C03611=1038.223,237.560,-108.650,170.961,41.926,157.985
C03612=1038.230,237.808,-108.678,170.964,41.928,157.986
C03613=1038.236,238.056,-108.706,170.967,41.929,157.986
C03614=1038.243,238.304,-108.734,170.970,41.930,157.987
C03615=1038.249,238.553,-108.763,170.972,41.931,157.987
C03616=1038.257,238.801,-108.791,170.975,41.933,157.988
C03617=1038.263,239.050,-108.819,170.978,41.934,157.988
C03618=1038.270,239.298,-108.848,170.981,41.935,157.988
C03619=1038.276,239.546,-108.876,170.983,41.936,157.989
C03620=1038.283,239.794,-108.904,170.987,41.937,157.989
C03621=1038.289,240.043,-108.933,170.989,41.938,157.990
C03622=1038.297,240.291,-108.961,170.992,41.940,157.990
C03623=1038.304,240.539,-108.990,170.994,41.941,157.990
C03624=1038.310,240.788,-109.018,170.998,41.942,157.991
C03625=1038.317,241.036,-109.047,171.000,41.943,157.991
C03626=1038.323,241.284,-109.076,171.003,41.945,157.992
C03627=1038.330,241.532,-109.103,171.005,41.946,157.992
C03628=1038.337,241.781,-109.133,171.009,41.947,157.993
C03629=1038.343,242.029,-109.162,171.012,41.949,157.993
C03630=1038.350,242.278,-109.190,171.014,41.950,157.994
C03631=1038.356,242.526,-109.219,171.016,41.951,157.994
C03632=1038.363,242.774,-109.247,171.020,41.952,157.994
C03633=1038.369,243.022,-109.276,171.022,41.954,157.995
C03634=1038.376,243.271,-109.304,171.025,41.955,157.995
C03635=1038.383,243.519,-109.333,171.028,41.956,157.996
C03636=1038.389,243.767,-109.362,171.031,41.958,157.996
C03637=1038.396,244.015,-109.391,171.033,41.959,157.997
C03638=1038.402,244.263,-109.420,171.037,41.960,157.997
C03639=1038.409,244.512,-109.448,171.040,41.962,157.998
C03640=1038.416,244.760,-109.477,171.042,41.963,157.998
C03641=1038.423,245.008,-109.505,171.045,41.964,157.999
C03642=1038.429,245.256,-109.534,171.048,41.965,157.999
C03643=1038.436,245.505,-109.564,171.051,41.966,157.999
C03644=1038.442,245.753,-109.593,171.053,41.968,158.000
C03645=1038.448,246.001,-109.622,171.057,41.969,158.001
C03646=1038.454,246.250,-109.651,171.059,41.970,158.001
C03647=1038.461,246.497,-109.679,171.062,41.972,158.001
C03648=1038.468,246.746,-109.709,171.065,41.973,158.002
C03649=1038.474,246.994,-109.738,171.068,41.974,158.002
C03650=1038.481,247.242,-109.767,171.070,41.976,158.003
C03651=1038.487,247.491,-109.796,171.074,41.977,158.003
C03652=1038.494,247.739,-109.825,171.077,41.979,158.004
C03653=1038.501,247.987,-109.854,171.079,41.980,158.004
C03654=1038.507,248.235,-109.883,171.083,41.981,158.005
C03655=1038.515,248.549,-109.920,171.085,41.983,158.005
C03656=1038.524,248.863,-109.957,171.089,41.985,158.006
C03657=1038.532,249.178,-109.993,171.092,41.986,158.006
C03658=1038.541,249.493,-110.030,171.096,41.988,158.007
C03659=1038.547,249.741,-110.059,171.100,41.989,158.007
C03660=1038.553,249.989,-110.088,171.102,41.991,158.008
C03661=1038.560,250.237,-110.119,171.105,41.992,158.008
C03662=1038.566,250.485,-110.148,171.108,41.994,158.009
C03663=1038.573,250.733,-110.177,171.111,41.995,158.009
C03664=1038.579,250.981,-110.206,171.114,41.996,158.010
C03665=1038.587,251.230,-110.235,171.117,41.998,158.010
C03666=1038.593,251.478,-110.264,171.119,41.998,158.011
C03667=1038.600,251.726,-110.294,171.123,42.000,158.011
C03668=1038.606,251.974,-110.323,171.126,42.001,158.012
C03669=1038.612,252.223,-110.352,171.129,42.003,158.012
C03670=1038.619,252.471,-110.381,171.132,42.004,158.013
C03671=1038.626,252.719,-110.411,171.134,42.005,158.013
C03672=1038.633,252.967,-110.439,171.138,42.007,158.014
C03673=1038.640,253.216,-110.469,171.140,42.008,158.014
C03674=1038.646,253.463,-110.499,171.144,42.009,158.015
C03675=1038.653,253.712,-110.528,171.146,42.011,158.015
C03676=1038.659,253.960,-110.557,171.149,42.012,158.016
C03677=1038.666,254.208,-110.586,171.152,42.013,158.016
C03678=1038.673,254.456,-110.616,171.155,42.015,158.016
C03679=1038.679,254.705,-110.645,171.159,42.016,158.017
C03680=1038.686,254.953,-110.675,171.161,42.018,158.017
C03681=1038.693,255.201,-110.704,171.165,42.018,158.018
C03682=1038.700,255.449,-110.733,171.167,42.020,158.018
C03683=1038.707,255.697,-110.763,171.171,42.021,158.019
C03684=1038.713,255.946,-110.792,171.173,42.023,158.019
C03685=1038.720,256.194,-110.821,171.176,42.024,158.020
C03686=1038.727,256.442,-110.852,171.179,42.025,158.020
C03687=1038.733,256.690,-110.881,171.182,42.027,158.021
C03688=1038.740,256.938,-110.911,171.186,42.028,158.021
C03689=1038.746,257.187,-110.940,171.188,42.029,158.022
C03690=1038.754,257.435,-110.970,171.192,42.031,158.022
C03691=1038.761,257.683,-110.998,171.194,42.032,158.023
C03692=1038.768,257.931,-111.028,171.198,42.033,158.023
C03693=1038.774,258.179,-111.057,171.200,42.034,158.024
C03694=1038.781,258.427,-111.088,171.204,42.036,158.024
C03695=1038.787,258.675,-111.117,171.206,42.037,158.025
C03696=1038.795,258.924,-111.147,171.210,42.038,158.025
C03697=1038.801,259.172,-111.176,171.212,42.040,158.026
C03698=1038.808,259.420,-111.206,171.216,42.041,158.026
C03699=1038.815,259.669,-111.235,171.219,42.043,158.027
C03700=1038.821,259.916,-111.265,171.222,42.044,158.027
C03701=1038.829,260.164,-111.295,171.225,42.045,158.027
C03702=1038.835,260.413,-111.324,171.228,42.046,158.028
C03703=1038.843,260.660,-111.354,171.232,42.048,158.029
C03704=1038.849,260.909,-111.383,171.234,42.049,158.029
C03705=1038.856,261.157,-111.413,171.238,42.050,158.029
C03706=1038.863,261.405,-111.443,171.240,42.052,158.030
C03707=1038.869,261.653,-111.472,171.244,42.053,158.030
C03708=1038.877,261.901,-111.502,171.246,42.055,158.031
C03709=1038.884,262.150,-111.532,171.250,42.056,158.032
C03710=1038.890,262.397,-111.563,171.253,42.058,158.032
C03711=1038.898,262.711,-111.600,171.256,42.059,158.033
C03712=1038.906,263.023,-111.638,171.261,42.061,158.033
C03713=1038.915,263.336,-111.676,171.265,42.063,158.034
C03714=1038.923,263.649,-111.713,171.268,42.064,158.034
C03715=1038.930,263.897,-111.744,171.272,42.066,158.035
C03716=1038.936,264.145,-111.774,171.275,42.067,158.036
C03717=1038.943,264.393,-111.804,171.278,42.069,158.036
C03718=1038.950,264.641,-111.834,171.281,42.070,158.037
C03719=1038.956,264.889,-111.865,171.284,42.072,158.037
C03720=1038.963,265.137,-111.895,171.287,42.073,158.038
C03721=1038.971,265.385,-111.925,171.291,42.075,158.038
C03722=1038.976,265.633,-111.955,171.293,42.076,158.039
C03723=1038.984,265.881,-111.985,171.297,42.077,158.039
C03724=1038.991,266.130,-112.015,171.300,42.079,158.040
C03725=1038.997,266.378,-112.046,171.303,42.080,158.040
C03726=1039.004,266.626,-112.076,171.307,42.082,158.041
C03727=1039.011,266.874,-112.106,171.309,42.083,158.041
C03728=1039.017,267.122,-112.136,171.313,42.085,158.042
C03729=1039.024,267.370,-112.166,171.316,42.086,158.042
C03730=1039.031,267.618,-112.197,171.319,42.088,158.043
C03731=1039.037,267.866,-112.227,171.323,42.089,158.043
C03732=1039.044,268.114,-112.257,171.325,42.091,158.044
C03733=1039.050,268.363,-112.288,171.329,42.092,158.044
C03734=1039.057,268.610,-112.317,171.332,42.093,158.045
C03735=1039.064,268.858,-112.349,171.335,42.095,158.045
C03736=1039.071,269.106,-112.379,171.339,42.096,158.046
C03737=1039.077,269.354,-112.409,171.341,42.098,158.046
C03738=1039.084,269.602,-112.440,171.345,42.099,158.047
C03739=1039.090,269.851,-112.470,171.348,42.101,158.048
C03740=1039.098,270.099,-112.501,171.351,42.102,158.048
C03741=1039.103,270.346,-112.531,171.355,42.104,158.049
C03742=1039.111,270.595,-112.562,171.357,42.106,158.049
C03743=1039.118,270.843,-112.592,171.361,42.107,158.050
C03744=1039.124,271.091,-112.623,171.365,42.109,158.050
C03745=1039.131,271.339,-112.654,171.367,42.110,158.051
C03746=1039.137,271.587,-112.684,171.371,42.111,158.051
C03747=1039.144,271.835,-112.715,171.374,42.113,158.052
C03748=1039.151,272.083,-112.745,171.377,42.114,158.052
C03749=1039.158,272.331,-112.776,171.381,42.116,158.053
C03750=1039.164,272.579,-112.807,171.384,42.118,158.054
C03751=1039.171,272.827,-112.837,171.387,42.119,158.054
C03752=1039.178,273.075,-112.868,171.391,42.121,158.055
C03753=1039.184,273.323,-112.899,171.394,42.122,158.055
C03754=1039.191,273.571,-112.929,171.397,42.124,158.056
C03755=1039.197,273.819,-112.960,171.401,42.125,158.056
C03756=1039.204,274.067,-112.991,171.404,42.127,158.057
C03757=1039.211,274.315,-113.022,171.407,42.129,158.057
C03758=1039.218,274.563,-113.053,171.411,42.130,158.058
C03759=1039.224,274.811,-113.084,171.414,42.131,158.059
C03760=1039.231,275.059,-113.114,171.417,42.133,158.059
C03761=1039.238,275.307,-113.145,171.421,42.135,158.060
C03762=1039.244,275.555,-113.176,171.424,42.136,158.060
C03763=1039.252,275.803,-113.207,171.427,42.138,158.061
C03764=1039.258,276.051,-113.238,171.430,42.139,158.061
C03765=1039.265,276.299,-113.269,171.434,42.141,158.062
C03766=1039.272,276.547,-113.300,171.437,42.143,158.063
C03767=1039.280,276.864,-113.340,171.442,42.145,158.063
C03768=1039.289,277.181,-113.380,171.445,42.147,158.064
C03769=1039.297,277.499,-113.418,171.450,42.148,158.065
C03770=1039.306,277.816,-113.458,171.454,42.150,158.065
C03771=1039.313,278.064,-113.490,171.458,42.152,158.066
C03772=1039.320,278.312,-113.521,171.461,42.154,158.067
C03773=1039.326,278.560,-113.552,171.465,42.155,158.067
C03774=1039.333,278.809,-113.583,171.468,42.157,158.068
C03775=1039.340,279.056,-113.614,171.471,42.159,158.068
C03776=1039.347,279.304,-113.645,171.475,42.160,158.069
C03777=1039.354,279.552,-113.677,171.478,42.162,158.069
C03778=1039.360,279.799,-113.708,171.481,42.164,158.070
C03779=1039.366,280.048,-113.739,171.485,42.165,158.071
C03780=1039.373,280.296,-113.770,171.489,42.167,158.071
C03781=1039.380,280.543,-113.801,171.491,42.168,158.072
C03782=1039.386,280.791,-113.833,171.495,42.170,158.072
C03783=1039.393,281.039,-113.864,171.499,42.172,158.073
C03784=1039.400,281.287,-113.896,171.502,42.173,158.074
C03785=1039.407,281.535,-113.927,171.505,42.175,158.074
C03786=1039.413,281.783,-113.959,171.509,42.177,158.075
C03787=1039.420,282.031,-113.990,171.513,42.179,158.075
C03788=1039.427,282.279,-114.022,171.516,42.180,158.076
C03789=1039.433,282.527,-114.053,171.520,42.181,158.076
C03790=1039.440,282.775,-114.084,171.523,42.184,158.077
C03791=1039.447,283.022,-114.116,171.526,42.185,158.078
C03792=1039.454,283.270,-114.147,171.530,42.187,158.078
C03793=1039.460,283.518,-114.179,171.534,42.188,158.079
C03794=1039.467,283.766,-114.210,171.536,42.190,158.080
C03795=1039.474,284.014,-114.242,171.540,42.192,158.080
C03796=1039.481,284.262,-114.273,171.544,42.194,158.081
C03797=1039.487,284.510,-114.304,171.548,42.195,158.081
C03798=1039.494,284.758,-114.336,171.551,42.197,158.082
C03799=1039.501,285.006,-114.368,171.555,42.199,158.083
C03800=1039.508,285.254,-114.400,171.558,42.200,158.083
C03801=1039.515,285.502,-114.431,171.561,42.202,158.084
C03802=1039.522,285.750,-114.463,171.565,42.203,158.084
C03803=1039.528,285.997,-114.494,171.569,42.205,158.085
C03804=1039.535,286.245,-114.526,171.572,42.207,158.086
C03805=1039.542,286.493,-114.558,171.576,42.209,158.086
C03806=1039.549,286.740,-114.589,171.580,42.210,158.087
C03807=1039.556,286.989,-114.621,171.583,42.212,158.087
C03808=1039.562,287.237,-114.653,171.586,42.214,158.088
C03809=1039.569,287.485,-114.685,171.590,42.216,158.089
C03810=1039.576,287.733,-114.716,171.594,42.217,158.089
C03811=1039.583,287.980,-114.748,171.597,42.219,158.090
C03812=1039.589,288.228,-114.781,171.601,42.221,158.091
C03813=1039.596,288.476,-114.812,171.604,42.222,158.091
C03814=1039.603,288.724,-114.844,171.608,42.224,158.092
C03815=1039.610,288.972,-114.876,171.611,42.226,158.092
C03816=1039.617,289.220,-114.907,171.615,42.228,158.093
C03817=1039.623,289.467,-114.940,171.619,42.230,158.094
C03818=1039.630,289.715,-114.972,171.623,42.231,158.094
C03819=1039.637,289.962,-115.004,171.626,42.233,158.095
C03820=1039.644,290.210,-115.035,171.630,42.235,158.096
C03821=1039.651,290.459,-115.068,171.633,42.237,158.096
C03822=1039.657,290.707,-115.100,171.637,42.239,158.097
C03823=1039.666,291.035,-115.143,171.642,42.241,158.098
C03824=1039.676,291.365,-115.185,171.647,42.243,158.099
C03825=1039.684,291.694,-115.228,171.652,42.246,158.099
C03826=1039.693,292.023,-115.271,171.657,42.248,158.100
C03827=1039.700,292.271,-115.303,171.660,42.250,158.101
C03828=1039.707,292.519,-115.335,171.664,42.252,158.102
C03829=1039.713,292.767,-115.367,171.668,42.254,158.102
C03830=1039.720,293.015,-115.399,171.671,42.255,158.103
C03831=1039.728,293.262,-115.431,171.675,42.257,158.104
C03832=1039.734,293.510,-115.464,171.678,42.259,158.104
C03833=1039.741,293.757,-115.496,171.682,42.261,158.105
C03834=1039.748,294.006,-115.528,171.686,42.263,158.106
C03835=1039.755,294.254,-115.561,171.689,42.264,158.106
C03836=1039.762,294.501,-115.593,171.693,42.266,158.107
C03837=1039.768,294.748,-115.626,171.697,42.268,158.107
C03838=1039.775,294.997,-115.657,171.701,42.270,158.108
C03839=1039.782,295.245,-115.690,171.705,42.272,158.109
C03840=1039.789,295.492,-115.722,171.708,42.274,158.109
C03841=1039.796,295.740,-115.755,171.712,42.275,158.110
C03842=1039.802,295.988,-115.788,171.716,42.277,158.111
C03843=1039.808,296.235,-115.821,171.720,42.279,158.112
C03844=1039.815,296.483,-115.853,171.723,42.281,158.112
C03845=1039.822,296.731,-115.886,171.727,42.283,158.113
C03846=1039.828,296.979,-115.919,171.731,42.285,158.114
C03847=1039.835,297.226,-115.952,171.735,42.287,158.114
C03848=1039.842,297.474,-115.984,171.739,42.289,158.115
C03849=1039.849,297.722,-116.017,171.743,42.291,158.116
C03850=1039.855,297.969,-116.050,171.746,42.293,158.116
C03851=1039.862,298.218,-116.083,171.750,42.295,158.117
C03852=1039.868,298.465,-116.115,171.754,42.297,158.118
C03853=1039.875,298.713,-116.148,171.758,42.299,158.118
C03854=1039.882,298.961,-116.181,171.762,42.301,158.119
C03855=1039.889,299.208,-116.214,171.765,42.303,158.120
C03856=1039.896,299.456,-116.247,171.769,42.305,158.121
C03857=1039.903,299.703,-116.279,171.773,42.307,158.121
C03858=1039.909,299.951,-116.312,171.777,42.309,158.122
C03859=1039.916,300.199,-116.345,171.781,42.311,158.123
C03860=1039.922,300.447,-116.378,171.785,42.313,158.123
C03861=1039.929,300.695,-116.412,171.789,42.315,158.124
C03862=1039.936,300.942,-116.444,171.792,42.317,158.125
C03863=1039.943,301.189,-116.477,171.796,42.319,158.126
C03864=1039.949,301.438,-116.510,171.800,42.321,158.126
C03865=1039.956,301.685,-116.543,171.804,42.323,158.127
C03866=1039.963,301.933,-116.576,171.808,42.325,158.128
C03867=1039.970,302.180,-116.609,171.811,42.327,158.128
C03868=1039.977,302.428,-116.642,171.815,42.329,158.129
C03869=1039.984,302.675,-116.675,171.819,42.331,158.130
C03870=1039.990,302.924,-116.708,171.823,42.333,158.131
C03871=1039.997,303.171,-116.742,171.827,42.335,158.131
C03872=1040.005,303.419,-116.774,171.831,42.337,158.132
C03873=1040.011,303.666,-116.807,171.835,42.339,158.133
C03874=1040.018,303.914,-116.841,171.838,42.341,158.133
C03875=1040.025,304.162,-116.874,171.843,42.343,158.134
C03876=1040.032,304.409,-116.907,171.847,42.345,158.135
C03877=1040.039,304.657,-116.940,171.851,42.348,158.136
C03878=1040.046,304.904,-116.973,171.855,42.350,158.136
C03879=1040.055,305.250,-117.020,171.860,42.353,158.137
C03880=1040.065,305.596,-117.066,171.866,42.355,158.138
C03881=1040.075,305.942,-117.112,171.871,42.358,158.139
C03882=1040.084,306.288,-117.159,171.877,42.361,158.140
C03883=1040.091,306.536,-117.193,171.882,42.363,158.141
C03884=1040.099,306.783,-117.225,171.885,42.365,158.142
C03885=1040.106,307.031,-117.259,171.889,42.367,158.143
C03886=1040.113,307.279,-117.292,171.893,42.369,158.143
C03887=1040.119,307.526,-117.325,171.897,42.371,158.144
C03888=1040.126,307.774,-117.359,171.901,42.373,158.145
C03889=1040.133,308.021,-117.393,171.905,42.375,158.146
C03890=1040.140,308.270,-117.426,171.910,42.377,158.146
C03891=1040.148,308.516,-117.459,171.914,42.380,158.147
C03892=1040.155,308.764,-117.493,171.917,42.382,158.148
C03893=1040.162,309.012,-117.526,171.921,42.384,158.149
C03894=1040.168,309.259,-117.559,171.925,42.386,158.149
C03895=1040.176,309.507,-117.593,171.930,42.388,158.150
C03896=1040.183,309.755,-117.627,171.934,42.390,158.151
C03897=1040.191,310.002,-117.660,171.938,42.392,158.152
C03898=1040.197,310.250,-117.693,171.942,42.394,158.152
C03899=1040.204,310.497,-117.727,171.947,42.396,158.153
C03900=1040.211,310.745,-117.760,171.951,42.398,158.154
C03901=1040.219,310.993,-117.794,171.955,42.401,158.155
C03902=1040.226,311.240,-117.828,171.958,42.403,158.155
C03903=1040.233,311.488,-117.862,171.962,42.405,158.156
C03904=1040.240,311.735,-117.895,171.967,42.407,158.157
C03905=1040.248,311.982,-117.929,171.971,42.409,158.158
C03906=1040.254,312.231,-117.962,171.975,42.411,158.159
C03907=1040.261,312.478,-117.997,171.979,42.413,158.159
C03908=1040.268,312.726,-118.031,171.984,42.416,158.160
C03909=1040.274,312.973,-118.065,171.988,42.418,158.161
C03910=1040.281,313.221,-118.098,171.992,42.420,158.162
C03911=1040.288,313.469,-118.133,171.996,42.423,158.163
C03912=1040.295,313.716,-118.167,172.000,42.425,158.163
C03913=1040.301,313.963,-118.201,172.005,42.427,158.164
C03914=1040.309,314.211,-118.235,172.009,42.430,158.165
C03915=1040.315,314.459,-118.270,172.013,42.432,158.166
C03916=1040.322,314.706,-118.304,172.017,42.434,158.167
C03917=1040.330,314.953,-118.338,172.022,42.436,158.167
C03918=1040.336,315.201,-118.372,172.026,42.439,158.168
C03919=1040.343,315.448,-118.406,172.030,42.441,158.169
C03920=1040.349,315.696,-118.440,172.034,42.443,158.170
C03921=1040.357,315.943,-118.475,172.039,42.446,158.171
C03922=1040.363,316.191,-118.509,172.043,42.448,158.172
C03923=1040.371,316.438,-118.544,172.047,42.451,158.172
C03924=1040.377,316.686,-118.578,172.050,42.453,158.173
C03925=1040.384,316.934,-118.612,172.056,42.455,158.174
C03926=1040.391,317.181,-118.647,172.060,42.458,158.175
C03927=1040.398,317.428,-118.681,172.064,42.460,158.176
C03928=1040.404,317.676,-118.716,172.068,42.462,158.177
C03929=1040.412,317.923,-118.750,172.072,42.464,158.177
C03930=1040.418,318.171,-118.784,172.077,42.467,158.178
C03931=1040.426,318.418,-118.819,172.082,42.469,158.179
C03932=1040.432,318.666,-118.853,172.086,42.472,158.180
C03933=1040.440,318.914,-118.888,172.090,42.474,158.181
C03934=1040.446,319.161,-118.923,172.093,42.476,158.182
C03935=1040.457,319.512,-118.972,172.100,42.480,158.183
C03936=1040.467,319.862,-119.020,172.106,42.483,158.184
C03937=1040.477,320.213,-119.069,172.113,42.487,158.185
C03938=1040.487,320.563,-119.118,172.118,42.490,158.186
C03939=1040.494,320.811,-119.153,172.123,42.492,158.187
C03940=1040.501,321.058,-119.187,172.127,42.495,158.188
C03941=1040.508,321.306,-119.222,172.132,42.497,158.189
C03942=1040.515,321.553,-119.257,172.136,42.500,158.190
C03943=1040.522,321.801,-119.291,172.141,42.502,158.191
C03944=1040.530,322.049,-119.326,172.146,42.505,158.192
C03945=1040.536,322.296,-119.361,172.150,42.507,158.193
C03946=1040.543,322.543,-119.396,172.155,42.510,158.193
C03947=1040.550,322.791,-119.430,172.159,42.512,158.194
C03948=1040.557,323.038,-119.465,172.163,42.515,158.195
C03949=1040.565,323.286,-119.500,172.168,42.517,158.196
C03950=1040.572,323.533,-119.535,172.172,42.519,158.197
C03951=1040.580,323.780,-119.570,172.177,42.522,158.198
C03952=1040.586,324.028,-119.604,172.181,42.524,158.199
C03953=1040.593,324.276,-119.639,172.185,42.527,158.199
C03954=1040.601,324.524,-119.674,172.190,42.529,158.200
C03955=1040.608,324.771,-119.709,172.194,42.532,158.201
C03956=1040.615,325.018,-119.744,172.199,42.534,158.202
C03957=1040.622,325.265,-119.779,172.203,42.537,158.203
C03958=1040.630,325.513,-119.814,172.208,42.539,158.204
C03959=1040.637,325.760,-119.849,172.212,42.541,158.205
C03960=1040.644,326.008,-119.883,172.217,42.544,158.206
C03961=1040.652,326.256,-119.919,172.222,42.547,158.207
C03962=1040.659,326.503,-119.954,172.227,42.549,158.208
C03963=1040.666,326.750,-119.989,172.231,42.552,158.208
C03964=1040.674,326.998,-120.024,172.236,42.554,158.209
C03965=1040.681,327.245,-120.059,172.240,42.557,158.210
C03966=1040.688,327.493,-120.094,172.245,42.559,158.211
C03967=1040.696,327.740,-120.129,172.249,42.562,158.212
C03968=1040.702,327.988,-120.164,172.254,42.564,158.213
C03969=1040.710,328.234,-120.199,172.258,42.567,158.214
C03970=1040.718,328.482,-120.235,172.263,42.569,158.215
C03971=1040.724,328.729,-120.270,172.267,42.572,158.216
C03972=1040.733,328.977,-120.305,172.273,42.575,158.217
C03973=1040.740,329.224,-120.341,172.277,42.577,158.218
C03974=1040.746,329.471,-120.376,172.282,42.580,158.219
C03975=1040.754,329.719,-120.411,172.286,42.583,158.219
C03976=1040.761,329.966,-120.447,172.291,42.585,158.220
C03977=1040.768,330.214,-120.482,172.295,42.588,158.221
C03978=1040.775,330.461,-120.518,172.300,42.590,158.222
C03979=1040.782,330.708,-120.554,172.306,42.593,158.223
C03980=1040.789,330.956,-120.589,172.310,42.596,158.224
C03981=1040.796,331.203,-120.625,172.315,42.599,158.225
C03982=1040.804,331.451,-120.660,172.319,42.601,158.226
C03983=1040.811,331.698,-120.696,172.324,42.604,158.227
C03984=1040.818,331.945,-120.731,172.328,42.607,158.228
C03985=1040.825,332.193,-120.768,172.334,42.609,158.229
C03986=1040.832,332.440,-120.803,172.338,42.613,158.230
C03987=1040.840,332.688,-120.839,172.343,42.615,158.231
C03988=1040.847,332.934,-120.875,172.348,42.618,158.232
C03989=1040.854,333.182,-120.910,172.352,42.620,158.233
C03990=1040.861,333.429,-120.946,172.357,42.623,158.234
C03991=1040.871,333.775,-120.997,172.364,42.627,158.235
C03992=1040.882,334.121,-121.047,172.371,42.631,158.237
C03993=1040.892,334.467,-121.096,172.377,42.634,158.238
C03994=1040.902,334.813,-121.147,172.384,42.638,158.239
C03995=1040.910,335.060,-121.183,172.389,42.641,158.240
C03996=1040.917,335.307,-121.219,172.394,42.644,158.241
C03997=1040.925,335.554,-121.255,172.399,42.647,158.243
C03998=1040.931,335.802,-121.290,172.404,42.650,158.243
C03999=1040.938,336.050,-121.327,172.408,42.653,158.244
C04000=1040.946,336.297,-121.363,172.413,42.656,158.245
C04001=1040.953,336.544,-121.399,172.419,42.659,158.247
C04002=1040.961,336.791,-121.435,172.423,42.662,158.248
C04003=1040.967,337.038,-121.472,172.428,42.664,158.249
C04004=1040.975,337.286,-121.508,172.432,42.667,158.250
C04005=1040.983,337.533,-121.544,172.438,42.670,158.251
C04006=1040.989,337.780,-121.581,172.443,42.673,158.252
C04007=1040.997,338.028,-121.617,172.448,42.676,158.253
C04008=1041.004,338.275,-121.653,172.452,42.679,158.254
C04009=1041.011,338.522,-121.689,172.458,42.682,158.255
C04010=1041.019,338.769,-121.727,172.463,42.685,158.256
C04011=1041.026,339.016,-121.763,172.467,42.688,158.257
C04012=1041.034,339.264,-121.799,172.473,42.691,158.258
C04013=1041.041,339.511,-121.835,172.478,42.693,158.259
C04014=1041.048,339.758,-121.872,172.482,42.697,158.260
C04015=1041.056,340.006,-121.908,172.487,42.699,158.261
C04016=1041.064,340.253,-121.945,172.493,42.702,158.262
C04017=1041.070,340.500,-121.981,172.498,42.705,158.263
C04018=1041.078,340.747,-122.017,172.502,42.708,158.264
C04019=1041.085,340.995,-122.054,172.507,42.711,158.265
C04020=1041.093,341.241,-122.091,172.513,42.714,158.266
C04021=1041.100,341.489,-122.127,172.518,42.717,158.267
C04022=1041.107,341.736,-122.163,172.524,42.720,158.269
C04023=1041.114,341.983,-122.201,172.528,42.723,158.270
C04024=1041.122,342.230,-122.237,172.533,42.726,158.271
C04025=1041.129,342.478,-122.275,172.538,42.729,158.272
C04026=1041.137,342.725,-122.311,172.544,42.732,158.273
C04027=1041.144,342.972,-122.348,172.548,42.736,158.274
C04028=1041.151,343.219,-122.384,172.553,42.739,158.275
C04029=1041.159,343.466,-122.422,172.559,42.742,158.276
C04030=1041.166,343.714,-122.458,172.564,42.745,158.277
C04031=1041.174,343.961,-122.495,172.570,42.748,158.278
C04032=1041.182,344.207,-122.532,172.574,42.751,158.279
C04033=1041.188,344.455,-122.569,172.579,42.754,158.281
C04034=1041.196,344.702,-122.606,172.585,42.757,158.282
C04035=1041.204,344.949,-122.644,172.590,42.760,158.283
C04036=1041.211,345.197,-122.680,172.595,42.764,158.284
C04037=1041.219,345.444,-122.717,172.601,42.767,158.285
C04038=1041.226,345.691,-122.755,172.605,42.770,158.286
C04039=1041.234,345.938,-122.792,172.610,42.773,158.287
C04040=1041.241,346.185,-122.829,172.616,42.777,158.289
C04041=1041.248,346.433,-122.866,172.621,42.779,158.290
C04042=1041.256,346.679,-122.903,172.627,42.783,158.291
C04043=1041.263,346.927,-122.941,172.632,42.786,158.292
C04044=1041.271,347.174,-122.978,172.638,42.789,158.293
C04045=1041.278,347.421,-123.015,172.642,42.792,158.294
C04046=1041.286,347.668,-123.053,172.647,42.796,158.295
C04047=1041.296,348.010,-123.104,172.655,42.800,158.297
C04048=1041.306,348.352,-123.155,172.662,42.805,158.299
C04049=1041.317,348.694,-123.207,172.670,42.809,158.300
C04050=1041.328,349.036,-123.259,172.677,42.813,158.302
C04051=1041.335,349.283,-123.297,172.683,42.817,158.303
C04052=1041.343,349.530,-123.334,172.688,42.820,158.304
C04053=1041.350,349.777,-123.371,172.693,42.823,158.305
C04054=1041.357,350.024,-123.409,172.699,42.827,158.306
C04055=1041.365,350.272,-123.446,172.704,42.830,158.308
C04056=1041.373,350.519,-123.484,172.710,42.833,158.309
C04057=1041.380,350.766,-123.522,172.715,42.837,158.310
C04058=1041.388,351.013,-123.559,172.721,42.840,158.311
C04059=1041.395,351.260,-123.597,172.726,42.843,158.312
C04060=1041.403,351.507,-123.634,172.732,42.847,158.314
C04061=1041.410,351.754,-123.673,172.737,42.850,158.315
C04062=1041.418,352.001,-123.711,172.743,42.854,158.316
C04063=1041.425,352.249,-123.748,172.748,42.857,158.317
C04064=1041.433,352.495,-123.786,172.754,42.860,158.319
C04065=1041.440,352.742,-123.824,172.759,42.864,158.320
C04066=1041.448,352.989,-123.862,172.765,42.867,158.321
C04067=1041.455,353.237,-123.900,172.770,42.871,158.322
C04068=1041.464,353.483,-123.938,172.776,42.874,158.324
C04069=1041.471,353.730,-123.975,172.781,42.878,158.325
C04070=1041.479,353.977,-124.014,172.787,42.881,158.326
C04071=1041.486,354.224,-124.051,172.793,42.885,158.327
C04072=1041.494,354.471,-124.089,172.798,42.888,158.328
C04073=1041.502,354.719,-124.127,172.804,42.891,158.330
C04074=1041.509,354.965,-124.166,172.809,42.895,158.331
C04075=1041.517,355.212,-124.204,172.815,42.899,158.332
C04076=1041.525,355.459,-124.242,172.820,42.902,158.334
C04077=1041.532,355.706,-124.280,172.826,42.906,158.335
C04078=1041.540,355.953,-124.319,172.831,42.909,158.336
C04079=1041.548,356.200,-124.356,172.837,42.913,158.337
C04080=1041.555,356.447,-124.394,172.844,42.916,158.339
C04081=1041.563,356.694,-124.433,172.849,42.920,158.340
C04082=1041.571,356.941,-124.471,172.855,42.923,158.341
C04083=1041.579,357.188,-124.510,172.860,42.927,158.343
C04084=1041.587,357.434,-124.548,172.866,42.931,158.344
C04085=1041.594,357.681,-124.586,172.872,42.934,158.345
C04086=1041.602,357.929,-124.624,172.877,42.938,158.346
C04087=1041.609,358.175,-124.662,172.883,42.942,158.348
C04088=1041.617,358.423,-124.702,172.890,42.945,158.349
C04089=1041.624,358.669,-124.740,172.895,42.949,158.350
C04090=1041.633,358.916,-124.779,172.901,42.953,158.352
C04091=1041.640,359.163,-124.817,172.906,42.956,158.353
C04092=1041.649,359.410,-124.856,172.912,42.960,158.354
C04093=1041.656,359.656,-124.894,172.919,42.963,158.356
C04094=1041.664,359.903,-124.933,172.924,42.967,158.357
C04095=1041.672,360.151,-124.972,172.930,42.971,158.358
C04096=1041.679,360.397,-125.010,172.936,42.975,158.360
C04097=1041.687,360.645,-125.049,172.941,42.978,158.361
C04098=1041.695,360.891,-125.087,172.948,42.982,158.362
C04099=1041.703,361.138,-125.127,172.954,42.986,158.364
C04100=1041.711,361.385,-125.166,172.959,42.990,158.365
C04101=1041.718,361.632,-125.204,172.965,42.994,158.366
C04102=1041.727,361.878,-125.243,172.972,42.997,158.368
C04103=1041.738,362.226,-125.298,172.980,43.003,158.370
C04104=1041.749,362.575,-125.353,172.989,43.008,158.372
C04105=1041.759,362.922,-125.409,172.997,43.014,158.374
C04106=1041.771,363.271,-125.463,173.006,43.019,158.376
C04107=1041.778,363.518,-125.503,173.011,43.023,158.377
C04108=1041.786,363.764,-125.541,173.017,43.027,158.378
C04109=1041.794,364.011,-125.581,173.023,43.031,158.380
C04110=1041.802,364.258,-125.620,173.030,43.035,158.381
C04111=1041.809,364.504,-125.659,173.035,43.039,158.383
C04112=1041.817,364.751,-125.699,173.041,43.043,158.384
C04113=1041.826,364.998,-125.737,173.048,43.046,158.385
C04114=1041.833,365.245,-125.777,173.054,43.050,158.387
C04115=1041.841,365.491,-125.816,173.059,43.054,158.388
C04116=1041.849,365.738,-125.856,173.066,43.058,158.390
C04117=1041.857,365.985,-125.895,173.072,43.062,158.391
C04118=1041.865,366.232,-125.935,173.078,43.066,158.392
C04119=1041.873,366.479,-125.974,173.085,43.070,158.394
C04120=1041.880,366.725,-126.014,173.091,43.074,158.395
C04121=1041.889,366.971,-126.053,173.097,43.078,158.397
C04122=1041.897,367.218,-126.093,173.103,43.082,158.398
C04123=1041.905,367.465,-126.132,173.109,43.086,158.400
C04124=1041.913,367.712,-126.172,173.116,43.090,158.401
C04125=1041.921,367.959,-126.211,173.122,43.094,158.403
C04126=1041.929,368.206,-126.251,173.128,43.098,158.404
C04127=1041.937,368.452,-126.291,173.134,43.103,158.406
C04128=1041.945,368.699,-126.331,173.141,43.107,158.407
C04129=1041.954,368.945,-126.370,173.147,43.110,158.409
C04130=1041.961,369.192,-126.410,173.153,43.115,158.410
C04131=1041.970,369.439,-126.449,173.160,43.119,158.412
C04132=1041.977,369.686,-126.489,173.166,43.123,158.413
C04133=1041.986,369.933,-126.528,173.173,43.127,158.415
C04134=1041.994,370.179,-126.568,173.179,43.132,158.416
C04135=1042.002,370.426,-126.609,173.185,43.135,158.418
C04136=1042.010,370.672,-126.648,173.191,43.140,158.419
C04137=1042.018,370.919,-126.688,173.198,43.144,158.421
C04138=1042.026,371.165,-126.729,173.204,43.148,158.422
C04139=1042.034,371.412,-126.769,173.211,43.153,158.424
C04140=1042.042,371.658,-126.809,173.217,43.157,158.425
C04141=1042.050,371.905,-126.849,173.224,43.161,158.427
C04142=1042.058,372.152,-126.889,173.230,43.165,158.428
C04143=1042.066,372.398,-126.929,173.237,43.170,158.430
C04144=1042.074,372.645,-126.970,173.244,43.174,158.432
C04145=1042.082,372.892,-127.010,173.250,43.179,158.433
C04146=1042.090,373.138,-127.050,173.257,43.182,158.435
C04147=1042.099,373.385,-127.090,173.263,43.187,158.436
C04148=1042.107,373.632,-127.131,173.270,43.191,158.438
C04149=1042.115,373.878,-127.171,173.276,43.196,158.439
C04150=1042.122,374.125,-127.211,173.283,43.200,158.441
C04151=1042.130,374.371,-127.252,173.290,43.204,158.443
C04152=1042.139,374.618,-127.293,173.296,43.209,158.444
C04153=1042.148,374.864,-127.333,173.303,43.213,158.446
C04154=1042.156,375.111,-127.373,173.309,43.218,158.447
C04155=1042.164,375.357,-127.413,173.316,43.222,158.449
C04156=1042.172,375.604,-127.454,173.323,43.226,158.451
C04157=1042.180,375.850,-127.495,173.329,43.231,158.452
C04158=1042.188,376.097,-127.536,173.336,43.236,158.454
C04159=1042.201,376.465,-127.596,173.346,43.242,158.456
C04160=1042.213,376.832,-127.657,173.357,43.249,158.459
C04161=1042.226,377.201,-127.718,173.367,43.256,158.461
C04162=1042.238,377.568,-127.779,173.377,43.262,158.464
C04163=1042.247,377.815,-127.820,173.384,43.267,158.466
C04164=1042.255,378.061,-127.860,173.391,43.271,158.467
C04165=1042.263,378.307,-127.901,173.397,43.276,158.469
C04166=1042.271,378.554,-127.942,173.404,43.280,158.471
C04167=1042.280,378.800,-127.983,173.412,43.285,158.472
C04168=1042.288,379.047,-128.024,173.419,43.290,158.474
C04169=1042.296,379.293,-128.065,173.425,43.295,158.476
C04170=1042.305,379.540,-128.107,173.432,43.299,158.477
C04171=1042.313,379.786,-128.147,173.439,43.304,158.479
C04172=1042.322,380.033,-128.188,173.446,43.309,158.481
C04173=1042.330,380.279,-128.230,173.454,43.313,158.483
C04174=1042.338,380.526,-128.271,173.460,43.318,158.484
C04175=1042.347,380.771,-128.312,173.467,43.323,158.486
C04176=1042.355,381.018,-128.353,173.474,43.327,158.488
C04177=1042.363,381.264,-128.395,173.481,43.332,158.489
C04178=1042.372,381.511,-128.437,173.489,43.337,158.491
C04179=1042.380,381.757,-128.478,173.496,43.342,158.493
C04180=1042.389,382.003,-128.519,173.502,43.347,158.495
C04181=1042.397,382.249,-128.561,173.510,43.352,158.497
C04182=1042.405,382.496,-128.602,173.517,43.356,158.498
C04183=1042.414,382.743,-128.644,173.524,43.361,158.500
C04184=1042.422,382.988,-128.686,173.531,43.366,158.502
C04185=1042.431,383.235,-128.727,173.539,43.371,158.504
C04186=1042.439,383.481,-128.770,173.546,43.376,158.506
C04187=1042.447,383.728,-128.810,173.553,43.381,158.507
C04188=1042.456,383.974,-128.852,173.561,43.385,158.509
C04189=1042.465,384.220,-128.894,173.568,43.390,158.511
C04190=1042.473,384.466,-128.936,173.575,43.395,158.513
C04191=1042.482,384.713,-128.977,173.582,43.400,158.515
C04192=1042.491,384.959,-129.019,173.590,43.405,158.516
C04193=1042.500,385.206,-129.061,173.597,43.410,158.518
C04194=1042.508,385.452,-129.103,173.605,43.415,158.520
C04195=1042.516,385.698,-129.144,173.612,43.420,158.522
C04196=1042.525,385.944,-129.186,173.619,43.425,158.524
C04197=1042.534,386.190,-129.229,173.627,43.430,158.526
C04198=1042.542,386.437,-129.271,173.634,43.435,158.528
C04199=1042.551,386.683,-129.313,173.642,43.440,158.529
C04200=1042.560,386.929,-129.354,173.649,43.445,158.531
C04201=1042.569,387.176,-129.397,173.656,43.450,158.533
C04202=1042.578,387.422,-129.439,173.664,43.455,158.535
C04203=1042.587,387.668,-129.481,173.671,43.460,158.537
C04204=1042.596,387.915,-129.522,173.679,43.465,158.539
C04205=1042.604,388.161,-129.565,173.686,43.471,158.541
C04206=1042.613,388.407,-129.607,173.693,43.476,158.543
C04207=1042.621,388.652,-129.650,173.701,43.481,158.545
C04208=1042.630,388.899,-129.692,173.710,43.486,158.547
C04209=1042.638,389.145,-129.735,173.717,43.491,158.548
C04210=1042.647,389.391,-129.776,173.724,43.496,158.550
C04211=1042.656,389.637,-129.819,173.732,43.502,158.552
C04212=1042.665,389.883,-129.862,173.740,43.507,158.554
C04213=1042.674,390.130,-129.904,173.747,43.512,158.556
C04214=1042.683,390.376,-129.947,173.756,43.518,158.558
C04215=1042.697,390.778,-130.017,173.768,43.526,158.562
C04216=1042.711,391.179,-130.087,173.781,43.535,158.565
C04217=1042.726,391.581,-130.156,173.793,43.544,158.568
C04218=1042.740,391.983,-130.226,173.806,43.552,158.571
C04219=1042.749,392.229,-130.269,173.814,43.558,158.573
C04220=1042.758,392.474,-130.311,173.822,43.564,158.575
C04221=1042.766,392.720,-130.354,173.830,43.569,158.577
C04222=1042.776,392.967,-130.398,173.838,43.574,158.579
C04223=1042.784,393.213,-130.441,173.846,43.579,158.581
C04224=1042.794,393.458,-130.484,173.853,43.585,158.584
C04225=1042.802,393.704,-130.527,173.862,43.591,158.586
C04226=1042.811,393.951,-130.570,173.870,43.596,158.588
C04227=1042.820,394.197,-130.613,173.877,43.602,158.590
C04228=1042.829,394.442,-130.656,173.886,43.607,158.592
C04229=1042.838,394.688,-130.699,173.894,43.613,158.594
C04230=1042.847,394.935,-130.743,173.903,43.618,158.596
C04231=1042.856,395.180,-130.786,173.910,43.624,158.598
C04232=1042.866,395.427,-130.829,173.918,43.630,158.600
C04233=1042.874,395.673,-130.873,173.927,43.635,158.602
C04234=1042.883,395.919,-130.916,173.935,43.641,158.605
C04235=1042.892,396.165,-130.960,173.943,43.646,158.607
C04236=1042.901,396.411,-131.003,173.951,43.652,158.609
C04237=1042.910,396.657,-131.047,173.960,43.658,158.611
C04238=1042.920,396.902,-131.091,173.968,43.664,158.613
C04239=1042.929,397.149,-131.134,173.976,43.670,158.615
C04240=1042.938,397.394,-131.178,173.984,43.675,158.618
C04241=1042.946,397.640,-131.221,173.992,43.681,158.620
C04242=1042.956,397.886,-131.265,174.001,43.687,158.622
C04243=1042.965,398.133,-131.309,174.009,43.693,158.624
C04244=1042.974,398.378,-131.353,174.018,43.698,158.626
C04245=1042.983,398.624,-131.397,174.027,43.704,158.628
C04246=1042.992,398.870,-131.441,174.034,43.710,158.631
C04247=1043.001,399.116,-131.485,174.044,43.716,158.633
C04248=1043.011,399.362,-131.529,174.051,43.722,158.635
C04249=1043.020,399.607,-131.573,174.060,43.728,158.637
C04250=1043.029,399.853,-131.617,174.069,43.734,158.640
C04251=1043.038,400.099,-131.661,174.077,43.740,158.642
C04252=1043.047,400.345,-131.704,174.086,43.745,158.644
C04253=1043.057,400.591,-131.749,174.094,43.752,158.646
C04254=1043.066,400.837,-131.793,174.103,43.757,158.649
C04255=1043.076,401.083,-131.838,174.112,43.764,158.651
C04256=1043.085,401.328,-131.881,174.120,43.769,158.653
C04257=1043.094,401.574,-131.925,174.129,43.776,158.656
C04258=1043.103,401.820,-131.969,174.138,43.782,158.658
C04259=1043.113,402.066,-132.014,174.146,43.788,158.660
C04260=1043.122,402.312,-132.059,174.155,43.794,158.663
C04261=1043.131,402.558,-132.104,174.164,43.800,158.665
C04262=1043.140,402.803,-132.148,174.173,43.806,158.667
C04263=1043.150,403.049,-132.192,174.181,43.812,158.670
C04264=1043.159,403.295,-132.236,174.191,43.819,158.672
C04265=1043.168,403.541,-132.282,174.200,43.825,158.674
C04266=1043.178,403.786,-132.327,174.209,43.831,158.677
C04267=1043.188,404.032,-132.371,174.218,43.837,158.679
C04268=1043.197,404.278,-132.416,174.226,43.844,158.682
C04269=1043.206,404.524,-132.461,174.235,43.850,158.684
C04270=1043.216,404.769,-132.506,174.244,43.856,158.686
C04271=1043.229,405.112,-132.569,174.257,43.865,158.690
C04272=1043.242,405.454,-132.632,174.269,43.874,158.693
C04273=1043.256,405.797,-132.694,174.283,43.882,158.697
C04274=1043.268,406.139,-132.757,174.295,43.892,158.700
C04275=1043.278,406.384,-132.801,174.305,43.898,158.703
C04276=1043.287,406.631,-132.847,174.314,43.904,158.705
C04277=1043.297,406.876,-132.892,174.323,43.911,158.708
C04278=1043.306,407.122,-132.938,174.333,43.917,158.710
C04279=1043.316,407.367,-132.983,174.342,43.924,158.713
C04280=1043.326,407.613,-133.028,174.351,43.930,158.715
C04281=1043.335,407.859,-133.074,174.360,43.937,158.718
C04282=1043.345,408.104,-133.119,174.370,43.943,158.720
C04283=1043.354,408.350,-133.165,174.379,43.950,158.723
C04284=1043.365,408.596,-133.210,174.389,43.957,158.725
C04285=1043.374,408.841,-133.256,174.398,43.963,158.728
C04286=1043.384,409.087,-133.301,174.407,43.970,158.730
C04287=1043.394,409.332,-133.347,174.417,43.976,158.733
C04288=1043.403,409.578,-133.392,174.426,43.983,158.736
C04289=1043.414,409.824,-133.438,174.436,43.990,158.738
C04290=1043.423,410.070,-133.483,174.445,43.997,158.741
C04291=1043.434,410.315,-133.529,174.456,44.003,158.743
C04292=1043.443,410.560,-133.575,174.465,44.010,158.746
C04293=1043.453,410.807,-133.621,174.474,44.016,158.749
C04294=1043.462,411.052,-133.667,174.484,44.024,158.751
C04295=1043.473,411.297,-133.713,174.495,44.030,158.754
C04296=1043.482,411.543,-133.759,174.504,44.037,158.757
C04297=1043.493,411.789,-133.804,174.514,44.044,158.759
C04298=1043.503,412.034,-133.850,174.523,44.050,158.762
C04299=1043.513,412.280,-133.896,174.534,44.057,158.765
C04300=1043.522,412.526,-133.943,174.543,44.064,158.767
C04301=1043.532,412.771,-133.989,174.553,44.071,158.770
C04302=1043.543,413.016,-134.035,174.564,44.078,158.773
C04303=1043.555,413.340,-134.097,174.577,44.088,158.777
C04304=1043.568,413.665,-134.158,174.589,44.097,158.780
C04305=1043.581,413.989,-134.219,174.603,44.106,158.784
C04306=1043.595,414.312,-134.281,174.616,44.116,158.788
C04307=1043.605,414.558,-134.327,174.627,44.123,158.790
C04308=1043.615,414.804,-134.373,174.637,44.130,158.793
C04309=1043.625,415.049,-134.420,174.647,44.137,158.796
C04310=1043.635,415.294,-134.466,174.657,44.144,158.799
C04311=1043.645,415.540,-134.514,174.668,44.151,158.802
C04312=1043.655,415.785,-134.561,174.678,44.158,158.805
C04313=1043.666,416.031,-134.607,174.688,44.165,158.807
C04314=1043.676,416.276,-134.654,174.698,44.173,158.810
C04315=1043.686,416.521,-134.701,174.709,44.180,158.813
C04316=1043.696,416.767,-134.748,174.719,44.188,158.816
C04317=1043.706,417.012,-134.795,174.730,44.194,158.819
C04318=1043.717,417.257,-134.842,174.741,44.202,158.822
C04319=1043.727,417.503,-134.889,174.751,44.209,158.825
C04320=1043.737,417.748,-134.936,174.762,44.216,158.828
C04321=1043.748,417.993,-134.983,174.773,44.224,158.831
C04322=1043.758,418.238,-135.030,174.783,44.232,158.834
C04323=1043.769,418.484,-135.078,174.793,44.238,158.836
C04324=1043.779,418.730,-135.125,174.804,44.246,158.839
C04325=1043.789,418.975,-135.172,174.815,44.254,158.843
C04326=1043.799,419.220,-135.220,174.826,44.261,158.846
C04327=1043.808,419.434,-135.261,174.835,44.268,158.848
C04328=1043.817,419.648,-135.302,174.845,44.274,158.851
C04329=1043.827,419.863,-135.344,174.854,44.281,158.854
C04330=1043.835,420.078,-135.386,174.864,44.287,158.856
C04331=1043.844,420.292,-135.428,174.873,44.295,158.859
C04332=1043.854,420.507,-135.469,174.883,44.301,158.862
C04333=1043.863,420.720,-135.511,174.892,44.307,158.864
C04334=1043.872,420.935,-135.553,174.902,44.315,158.867
C04335=1043.883,421.181,-135.601,174.913,44.322,158.870
C04336=1043.893,421.425,-135.649,174.925,44.330,158.873
C04337=1043.904,421.670,-135.697,174.936,44.337,158.876
C04338=1043.914,421.916,-135.744,174.947,44.345,158.879
C04339=1043.925,422.161,-135.792,174.958,44.353,158.883
C04340=1043.936,422.406,-135.840,174.970,44.361,158.886
C04341=1043.946,422.651,-135.889,174.981,44.368,158.889
C04342=1043.956,422.897,-135.936,174.992,44.376,158.892
C04343=1043.967,423.142,-135.984,175.003,44.384,158.895
C04344=1043.978,423.387,-136.033,175.015,44.392,158.898
C04345=1043.989,423.632,-136.081,175.026,44.400,158.902
C04346=1044.000,423.877,-136.129,175.037,44.408,158.905
C04347=1044.010,424.122,-136.177,175.050,44.416,158.908
C04348=1044.021,424.367,-136.226,175.061,44.424,158.912
C04349=1044.032,424.612,-136.275,175.072,44.432,158.915
C04350=1044.043,424.857,-136.323,175.084,44.440,158.918
C04351=1044.053,425.102,-136.371,175.095,44.448,158.921
C04352=1044.064,425.347,-136.421,175.108,44.456,158.925
C04353=1044.075,425.593,-136.469,175.119,44.464,158.928
C04354=1044.086,425.837,-136.518,175.131,44.472,158.931
C04355=1044.096,426.082,-136.566,175.143,44.481,158.935
C04356=1044.108,426.327,-136.615,175.155,44.489,158.938
C04357=1044.119,426.572,-136.664,175.166,44.497,158.941
C04358=1044.130,426.817,-136.713,175.179,44.505,158.945
C04359=1044.140,427.061,-136.762,175.191,44.513,158.948
C04360=1044.151,427.307,-136.811,175.202,44.522,158.952
C04361=1044.162,427.552,-136.860,175.215,44.530,158.955
C04362=1044.174,427.797,-136.909,175.227,44.539,158.959
C04363=1044.184,428.042,-136.959,175.240,44.547,158.962
C04364=1044.196,428.286,-137.008,175.251,44.555,158.966
C04365=1044.206,428.531,-137.057,175.264,44.563,158.969
C04366=1044.218,428.777,-137.107,175.276,44.572,158.973
C04367=1044.229,429.022,-137.156,175.288,44.580,158.976
C04368=1044.240,429.267,-137.205,175.301,44.589,158.980
C04369=1044.251,429.512,-137.255,175.313,44.598,158.983
C04370=1044.263,429.756,-137.304,175.326,44.606,158.987
C04371=1044.273,430.001,-137.354,175.338,44.615,158.990
C04372=1044.284,430.246,-137.404,175.351,44.623,158.994
C04373=1044.296,430.490,-137.453,175.364,44.632,158.998
C04374=1044.306,430.735,-137.503,175.377,44.641,159.001
C04375=1044.317,430.980,-137.553,175.389,44.649,159.005
C04376=1044.330,431.224,-137.603,175.401,44.658,159.009
C04377=1044.340,431.469,-137.653,175.414,44.667,159.012
C04378=1044.352,431.714,-137.703,175.428,44.676,159.016
C04379=1044.364,431.959,-137.753,175.441,44.684,159.020
C04380=1044.374,432.204,-137.803,175.453,44.693,159.023
C04381=1044.386,432.448,-137.853,175.466,44.702,159.027
C04382=1044.398,432.693,-137.903,175.479,44.711,159.031
C04383=1044.409,432.937,-137.954,175.492,44.720,159.035
C04384=1044.421,433.182,-138.004,175.505,44.729,159.038
C04385=1044.432,433.427,-138.054,175.518,44.738,159.042
C04386=1044.444,433.672,-138.105,175.532,44.747,159.046
C04387=1044.455,433.896,-138.151,175.544,44.755,159.049
C04388=1044.465,434.121,-138.197,175.556,44.763,159.053
C04389=1044.476,434.345,-138.244,175.569,44.771,159.057
C04390=1044.486,434.570,-138.290,175.581,44.780,159.060
C04391=1044.498,434.794,-138.336,175.594,44.788,159.064
C04392=1044.508,435.018,-138.383,175.605,44.796,159.067
C04393=1044.519,435.244,-138.430,175.618,44.805,159.071
C04394=1044.530,435.468,-138.476,175.631,44.814,159.074
C04395=1044.542,435.712,-138.527,175.644,44.823,159.078
C04396=1044.553,435.957,-138.578,175.658,44.832,159.082
C04397=1044.565,436.201,-138.629,175.672,44.841,159.086
C04398=1044.577,436.445,-138.680,175.685,44.850,159.090
C04399=1044.589,436.690,-138.731,175.700,44.860,159.094
C04400=1044.601,436.935,-138.782,175.713,44.869,159.098
C04401=1044.612,437.179,-138.833,175.727,44.878,159.102
C04402=1044.624,437.423,-138.884,175.741,44.888,159.106
C04403=1044.636,437.668,-138.936,175.755,44.897,159.110
C04404=1044.647,437.912,-138.987,175.770,44.907,159.115
C04405=1044.660,438.156,-139.039,175.783,44.916,159.119
C04406=1044.672,438.401,-139.091,175.798,44.926,159.123
C04407=1044.683,438.645,-139.142,175.812,44.935,159.127
C04408=1044.696,438.890,-139.193,175.826,44.945,159.131
C04409=1044.708,439.133,-139.245,175.841,44.954,159.135
C04410=1044.720,439.378,-139.297,175.855,44.964,159.140
C04411=1044.732,439.622,-139.349,175.870,44.974,159.144
C04412=1044.745,439.867,-139.400,175.885,44.984,159.148
C04413=1044.757,440.111,-139.453,175.898,44.993,159.152
C04414=1044.769,440.355,-139.504,175.913,45.003,159.157
C04415=1044.781,440.599,-139.556,175.928,45.013,159.161
C04416=1044.794,440.844,-139.609,175.943,45.022,159.165
C04417=1044.806,441.088,-139.661,175.958,45.033,159.170
C04418=1044.817,441.332,-139.713,175.973,45.042,159.174
C04419=1044.830,441.577,-139.766,175.988,45.052,159.178
C04420=1044.842,441.820,-139.818,176.002,45.062,159.183
C04421=1044.855,442.064,-139.870,176.017,45.072,159.187
C04422=1044.867,442.309,-139.923,176.033,45.082,159.192
C04423=1044.880,442.553,-139.975,176.049,45.092,159.196
C04424=1044.892,442.797,-140.027,176.064,45.102,159.201
C04425=1044.905,443.041,-140.080,176.079,45.112,159.205
C04426=1044.917,443.286,-140.133,176.094,45.122,159.209
C04427=1044.929,443.529,-140.186,176.109,45.132,159.214
C04428=1044.942,443.773,-140.238,176.125,45.143,159.219
C04429=1044.955,444.017,-140.292,176.140,45.153,159.223
C04430=1044.968,444.261,-140.344,176.157,45.163,159.228
C04431=1044.981,444.505,-140.397,176.172,45.174,159.232
C04432=1044.994,444.749,-140.450,176.187,45.184,159.237
C04433=1045.006,444.993,-140.503,176.204,45.194,159.242
C04434=1045.018,445.237,-140.556,176.219,45.204,159.246
C04435=1045.032,445.480,-140.609,176.236,45.215,159.251
C04436=1045.046,445.722,-140.661,176.251,45.225,159.255
C04437=1045.060,445.966,-140.712,176.267,45.235,159.260
C04438=1045.075,446.210,-140.764,176.284,45.245,159.265
C04439=1045.091,446.454,-140.814,176.300,45.255,159.269
C04440=1045.107,446.698,-140.865,176.316,45.264,159.274
C04441=1045.124,446.942,-140.915,176.333,45.274,159.278
C04442=1045.141,447.186,-140.964,176.349,45.284,159.283
C04443=1045.160,447.430,-141.013,176.365,45.293,159.287
C04444=1045.179,447.673,-141.061,176.382,45.302,159.292
C04445=1045.198,447.919,-141.110,176.399,45.311,159.296
C04446=1045.218,448.163,-141.156,176.415,45.320,159.300
C04447=1045.238,448.402,-141.202,176.432,45.328,159.305
C04448=1045.259,448.642,-141.248,176.449,45.337,159.309
C04449=1045.281,448.881,-141.292,176.466,45.346,159.313
C04450=1045.303,449.120,-141.337,176.482,45.354,159.318
C04451=1045.325,449.359,-141.381,176.499,45.362,159.322
C04452=1045.349,449.599,-141.424,176.516,45.370,159.326
C04453=1045.373,449.839,-141.466,176.532,45.378,159.330
C04454=1045.397,450.078,-141.509,176.550,45.386,159.334
C04455=1045.423,450.323,-141.552,176.567,45.394,159.338
C04456=1045.450,450.569,-141.594,176.584,45.401,159.343
C04457=1045.476,450.815,-141.636,176.602,45.409,159.347
C04458=1045.503,451.060,-141.678,176.619,45.417,159.351
C04459=1045.199,451.097,-141.988,176.621,45.500,159.376
C04460=1045.172,450.851,-141.946,176.604,45.493,159.372
C04461=1045.144,450.606,-141.904,176.586,45.485,159.368
C04462=1045.118,450.361,-141.862,176.568,45.477,159.363
C04463=1045.092,450.115,-141.819,176.551,45.470,159.359
C04464=1045.067,449.884,-141.779,176.534,45.462,159.355
C04465=1045.044,449.653,-141.737,176.518,45.455,159.351
C04466=1045.022,449.422,-141.695,176.502,45.447,159.347
C04467=1045.000,449.191,-141.653,176.485,45.439,159.343
C04468=1044.978,448.960,-141.610,176.470,45.431,159.339
C04469=1044.957,448.729,-141.567,176.453,45.423,159.335
C04470=1044.937,448.497,-141.524,176.437,45.415,159.331
C04471=1044.917,448.267,-141.480,176.421,45.407,159.327
C04472=1044.896,448.022,-141.432,176.404,45.398,159.322
C04473=1044.877,447.777,-141.385,176.388,45.389,159.318
C04474=1044.857,447.533,-141.338,176.370,45.380,159.313
C04475=1044.839,447.289,-141.288,176.354,45.371,159.309
C04476=1044.821,447.045,-141.239,176.337,45.361,159.304
C04477=1044.803,446.801,-141.190,176.321,45.352,159.300
C04478=1044.787,446.558,-141.140,176.305,45.342,159.295
C04479=1044.771,446.313,-141.089,176.289,45.333,159.291
C04480=1044.756,446.070,-141.039,176.272,45.323,159.286
C04481=1044.740,445.825,-140.987,176.256,45.314,159.282
C04482=1044.727,445.583,-140.935,176.239,45.303,159.277
C04483=1044.712,445.341,-140.883,176.224,45.293,159.272
C04484=1044.699,445.097,-140.830,176.207,45.283,159.268
C04485=1044.686,444.853,-140.776,176.192,45.273,159.263
C04486=1044.674,444.609,-140.724,176.176,45.263,159.259
C04487=1044.661,444.365,-140.671,176.160,45.252,159.254
C04488=1044.649,444.121,-140.618,176.145,45.242,159.249
C04489=1044.636,443.877,-140.565,176.128,45.232,159.245
C04490=1044.623,443.633,-140.512,176.113,45.222,159.240
C04491=1044.611,443.389,-140.459,176.098,45.212,159.236
C04492=1044.598,443.145,-140.407,176.082,45.202,159.231
C04493=1044.586,442.901,-140.354,176.067,45.192,159.227
C04494=1044.573,442.657,-140.301,176.051,45.182,159.222
C04495=1044.561,442.413,-140.249,176.036,45.172,159.218
C04496=1044.548,442.169,-140.196,176.021,45.162,159.213
C04497=1044.536,441.925,-140.143,176.005,45.152,159.209
C04498=1044.523,441.680,-140.091,175.990,45.142,159.204
C04499=1044.511,441.436,-140.039,175.975,45.132,159.200
C04500=1044.499,441.192,-139.987,175.960,45.122,159.196
C04501=1044.486,440.948,-139.934,175.945,45.112,159.191
C04502=1044.474,440.704,-139.882,175.930,45.103,159.187
C04503=1044.462,440.459,-139.831,175.916,45.093,159.183
C04504=1044.449,440.215,-139.778,175.901,45.083,159.178
C04505=1044.437,439.971,-139.726,175.887,45.074,159.174
C04506=1044.425,439.726,-139.675,175.872,45.064,159.170
C04507=1044.413,439.483,-139.622,175.857,45.054,159.166
C04508=1044.401,439.238,-139.571,175.843,45.045,159.161
C04509=1044.389,438.994,-139.519,175.828,45.035,159.157
C04510=1044.376,438.749,-139.467,175.813,45.026,159.153
C04511=1044.365,438.504,-139.416,175.800,45.016,159.149
C04512=1044.352,438.261,-139.364,175.785,45.007,159.145
C04513=1044.340,438.016,-139.312,175.771,44.997,159.141
C04514=1044.328,437.772,-139.261,175.757,44.988,159.136
C04515=1044.316,437.527,-139.210,175.743,44.979,159.132
C04516=1044.305,437.284,-139.159,175.728,44.969,159.128
C04517=1044.293,437.039,-139.108,175.715,44.960,159.124
C04518=1044.281,436.795,-139.056,175.700,44.950,159.120
C04519=1044.269,436.550,-139.005,175.687,44.941,159.116
C04520=1044.257,436.306,-138.953,175.672,44.932,159.112
C04521=1044.245,436.061,-138.903,175.659,44.923,159.108
C04522=1044.234,435.817,-138.852,175.645,44.914,159.104
C04523=1044.222,435.572,-138.801,175.631,44.905,159.100
C04524=1044.211,435.347,-138.754,175.619,44.896,159.097
C04525=1044.199,435.121,-138.707,175.606,44.888,159.093
C04526=1044.189,434.896,-138.660,175.594,44.880,159.089
C04527=1044.178,434.670,-138.614,175.581,44.871,159.086
C04528=1044.167,434.444,-138.567,175.568,44.863,159.082
C04529=1044.157,434.219,-138.521,175.556,44.854,159.079
C04530=1044.146,433.994,-138.474,175.543,44.846,159.075
C04531=1044.135,433.768,-138.427,175.532,44.838,159.072
C04532=1044.123,433.523,-138.377,175.518,44.829,159.068
C04533=1044.112,433.279,-138.327,175.505,44.820,159.064
C04534=1044.100,433.034,-138.276,175.492,44.811,159.060
C04535=1044.089,432.790,-138.226,175.479,44.802,159.056
C04536=1044.077,432.545,-138.175,175.466,44.794,159.053
C04537=1044.065,432.301,-138.126,175.452,44.785,159.049
C04538=1044.054,432.056,-138.075,175.439,44.776,159.045
C04539=1044.043,431.810,-138.025,175.426,44.768,159.041
C04540=1044.031,431.566,-137.976,175.413,44.759,159.038
C04541=1044.020,431.322,-137.925,175.400,44.750,159.034
C04542=1044.009,431.076,-137.875,175.387,44.741,159.030
C04543=1043.997,430.832,-137.826,175.375,44.733,159.027
C04544=1043.986,430.587,-137.775,175.362,44.724,159.023
C04545=1043.975,430.343,-137.726,175.349,44.715,159.019
C04546=1043.964,430.098,-137.676,175.336,44.707,159.016
C04547=1043.953,429.853,-137.626,175.325,44.698,159.012
C04548=1043.941,429.608,-137.577,175.312,44.690,159.009
C04549=1043.930,429.363,-137.527,175.299,44.682,159.005
C04550=1043.919,429.119,-137.478,175.287,44.673,159.001
C04551=1043.908,428.874,-137.428,175.274,44.665,158.998
C04552=1043.898,428.629,-137.378,175.261,44.656,158.994
C04553=1043.886,428.384,-137.329,175.250,44.648,158.991
C04554=1043.875,428.139,-137.280,175.237,44.640,158.987
C04555=1043.864,427.894,-137.231,175.225,44.631,158.984
C04556=1043.853,427.649,-137.182,175.212,44.623,158.980
C04557=1043.842,427.404,-137.132,175.201,44.614,158.977
C04558=1043.831,427.159,-137.083,175.188,44.606,158.974
C04559=1043.820,426.914,-137.035,175.176,44.598,158.970
C04560=1043.809,426.669,-136.985,175.164,44.590,158.967
C04561=1043.798,426.424,-136.936,175.152,44.582,158.963
C04562=1043.786,426.179,-136.888,175.141,44.574,158.960
C04563=1043.776,425.935,-136.839,175.128,44.565,158.957
C04564=1043.765,425.690,-136.790,175.117,44.558,158.953
C04565=1043.754,425.444,-136.741,175.105,44.549,158.950
C04566=1043.743,425.199,-136.693,175.093,44.542,158.947
C04567=1043.733,424.955,-136.644,175.081,44.533,158.943
C04568=1043.722,424.709,-136.596,175.070,44.525,158.940
C04569=1043.711,424.464,-136.547,175.058,44.517,158.937
C04570=1043.700,424.220,-136.498,175.046,44.509,158.933
C04571=1043.689,423.974,-136.450,175.034,44.501,158.930
C04572=1043.678,423.729,-136.401,175.023,44.494,158.927
C04573=1043.668,423.484,-136.354,175.011,44.486,158.924
C04574=1043.657,423.239,-136.305,175.000,44.478,158.920
C04575=1043.646,422.994,-136.257,174.989,44.470,158.917
C04576=1043.635,422.749,-136.209,174.976,44.462,158.914
C04577=1043.625,422.503,-136.160,174.965,44.455,158.911
C04578=1043.614,422.258,-136.113,174.954,44.447,158.908
C04579=1043.604,422.013,-136.065,174.943,44.439,158.904
C04580=1043.593,421.768,-136.017,174.931,44.431,158.901
C04581=1043.582,421.523,-135.969,174.920,44.424,158.898
C04582=1043.572,421.277,-135.921,174.909,44.416,158.895
C04583=1043.561,421.033,-135.873,174.898,44.409,158.892
C04584=1043.552,420.818,-135.831,174.888,44.402,158.889
C04585=1043.543,420.601,-135.789,174.878,44.395,158.887
C04586=1043.534,420.386,-135.747,174.869,44.389,158.884
C04587=1043.524,420.171,-135.705,174.859,44.382,158.881
C04588=1043.515,419.955,-135.664,174.850,44.375,158.878
C04589=1043.506,419.740,-135.622,174.840,44.369,158.876
C04590=1043.496,419.524,-135.580,174.830,44.362,158.873
C04591=1043.488,419.309,-135.537,174.821,44.356,158.870
C04592=1043.478,419.063,-135.490,174.810,44.348,158.867
C04593=1043.468,418.818,-135.443,174.799,44.341,158.864
C04594=1043.457,418.573,-135.396,174.789,44.333,158.861
C04595=1043.447,418.328,-135.349,174.778,44.326,158.858
C04596=1043.437,418.082,-135.301,174.767,44.318,158.855
C04597=1043.426,417.837,-135.255,174.756,44.311,158.852
C04598=1043.415,417.591,-135.207,174.746,44.304,158.850
C04599=1043.405,417.346,-135.160,174.735,44.296,158.847
C04600=1043.395,417.101,-135.113,174.724,44.289,158.844
C04601=1043.385,416.855,-135.065,174.714,44.282,158.841
C04602=1043.374,416.610,-135.018,174.703,44.275,158.838
C04603=1043.364,416.365,-134.972,174.692,44.267,158.835
C04604=1043.354,416.119,-134.925,174.683,44.260,158.832
C04605=1043.343,415.874,-134.878,174.672,44.253,158.829
C04606=1043.334,415.628,-134.831,174.662,44.246,158.826
C04607=1043.323,415.383,-134.784,174.651,44.239,158.824
C04608=1043.313,415.139,-134.738,174.641,44.232,158.821
C04609=1043.303,414.893,-134.691,174.630,44.225,158.818
C04610=1043.293,414.647,-134.644,174.621,44.218,158.815
C04611=1043.283,414.401,-134.598,174.610,44.211,158.812
C04612=1043.272,414.156,-134.552,174.600,44.204,158.810
C04613=1043.263,413.911,-134.505,174.590,44.197,158.807
C04614=1043.253,413.665,-134.458,174.580,44.190,158.804
C04615=1043.243,413.419,-134.412,174.569,44.183,158.801
C04616=1043.233,413.174,-134.365,174.559,44.175,158.798
C04617=1043.223,412.929,-134.319,174.550,44.169,158.796
C04618=1043.213,412.683,-134.273,174.539,44.162,158.793
C04619=1043.203,412.437,-134.226,174.529,44.155,158.790
C04620=1043.194,412.192,-134.180,174.520,44.148,158.787
C04621=1043.183,411.947,-134.134,174.509,44.141,158.785
C04622=1043.173,411.701,-134.088,174.500,44.135,158.782
C04623=1043.163,411.456,-134.042,174.490,44.128,158.779
C04624=1043.154,411.209,-133.996,174.480,44.121,158.777
C04625=1043.144,410.964,-133.951,174.470,44.114,158.774
C04626=1043.133,410.719,-133.905,174.461,44.108,158.771
C04627=1043.123,410.473,-133.858,174.451,44.101,158.769
C04628=1043.113,410.227,-133.814,174.440,44.094,158.766
C04629=1043.104,409.982,-133.767,174.431,44.087,158.763
C04630=1043.094,409.737,-133.722,174.422,44.081,158.761
C04631=1043.084,409.490,-133.676,174.412,44.074,158.758
C04632=1043.074,409.245,-133.630,174.403,44.068,158.756
C04633=1043.065,408.999,-133.585,174.393,44.061,158.753
C04634=1043.054,408.754,-133.539,174.384,44.055,158.751
C04635=1043.045,408.508,-133.494,174.374,44.048,158.748
C04636=1043.036,408.262,-133.449,174.364,44.042,158.745
C04637=1043.025,408.017,-133.403,174.355,44.035,158.743
C04638=1043.016,407.771,-133.357,174.346,44.029,158.740
C04639=1043.006,407.526,-133.313,174.336,44.022,158.738
C04640=1042.996,407.280,-133.267,174.327,44.016,158.735
C04641=1042.987,407.034,-133.221,174.318,44.009,158.733
C04642=1042.977,406.789,-133.176,174.308,44.003,158.730
C04643=1042.968,406.543,-133.131,174.299,43.997,158.728
C04644=1042.960,406.331,-133.092,174.291,43.991,158.726
C04645=1042.951,406.119,-133.054,174.283,43.986,158.724
C04646=1042.943,405.909,-133.015,174.275,43.980,158.721
C04647=1042.935,405.696,-132.976,174.268,43.975,158.719
C04648=1042.927,405.485,-132.937,174.260,43.969,158.717
C04649=1042.919,405.274,-132.898,174.251,43.964,158.715
C04650=1042.911,405.062,-132.859,174.243,43.958,158.713
C04651=1042.902,404.850,-132.821,174.236,43.953,158.711
C04652=1042.894,404.633,-132.780,174.228,43.947,158.709
C04653=1042.886,404.415,-132.741,174.220,43.942,158.707
C04654=1042.877,404.198,-132.701,174.212,43.936,158.704
C04655=1042.869,403.980,-132.662,174.204,43.930,158.702
C04656=1042.860,403.763,-132.622,174.195,43.925,158.700
C04657=1042.853,403.545,-132.582,174.188,43.920,158.698
C04658=1042.845,403.327,-132.543,174.180,43.914,158.696
C04659=1042.836,403.110,-132.503,174.172,43.909,158.694
C04660=1042.827,402.864,-132.459,174.163,43.903,158.692
C04661=1042.817,402.618,-132.414,174.154,43.897,158.689
C04662=1042.807,402.372,-132.370,174.146,43.890,158.687
C04663=1042.798,402.127,-132.325,174.137,43.885,158.685
C04664=1042.790,401.881,-132.280,174.128,43.879,158.682
C04665=1042.780,401.635,-132.236,174.119,43.872,158.680
C04666=1042.770,401.389,-132.191,174.111,43.867,158.678
C04667=1042.761,401.143,-132.147,174.102,43.860,158.675
C04668=1042.752,400.897,-132.103,174.093,43.855,158.673
C04669=1042.743,400.652,-132.059,174.085,43.848,158.671
C04670=1042.733,400.406,-132.015,174.076,43.843,158.668
C04671=1042.724,400.160,-131.971,174.067,43.837,158.666
C04672=1042.715,399.914,-131.927,174.059,43.831,158.664
C04673=1042.706,399.668,-131.883,174.050,43.825,158.662
C04674=1042.696,399.422,-131.839,174.041,43.820,158.659
C04675=1042.687,399.177,-131.795,174.033,43.813,158.657
C04676=1042.678,398.931,-131.751,174.024,43.807,158.655
C04677=1042.668,398.684,-131.707,174.016,43.802,158.653
C04678=1042.660,398.439,-131.663,174.007,43.796,158.650
C04679=1042.650,398.193,-131.619,173.998,43.790,158.648
C04680=1042.641,397.947,-131.575,173.990,43.785,158.646
C04681=1042.632,397.701,-131.531,173.982,43.779,158.644
C04682=1042.622,397.455,-131.488,173.974,43.773,158.642
C04683=1042.613,397.209,-131.444,173.965,43.767,158.639
C04684=1042.604,396.963,-131.400,173.957,43.761,158.637
C04685=1042.595,396.717,-131.357,173.948,43.756,158.635
C04686=1042.587,396.472,-131.314,173.940,43.750,158.633
C04687=1042.577,396.226,-131.269,173.932,43.745,158.631
C04688=1042.569,395.980,-131.226,173.924,43.739,158.629
C04689=1042.559,395.733,-131.182,173.915,43.733,158.626
C04690=1042.551,395.487,-131.139,173.907,43.728,158.624
C04691=1042.541,395.242,-131.096,173.899,43.722,158.622
C04692=1042.532,394.996,-131.053,173.891,43.716,158.620
C04693=1042.523,394.750,-131.009,173.883,43.711,158.618
C04694=1042.514,394.503,-130.966,173.874,43.705,158.616
C04695=1042.505,394.258,-130.923,173.867,43.700,158.614
C04696=1042.496,394.012,-130.879,173.859,43.695,158.612
C04697=1042.487,393.765,-130.836,173.850,43.689,158.610
C04698=1042.478,393.520,-130.794,173.842,43.684,158.608
C04699=1042.469,393.274,-130.751,173.834,43.678,158.605
C04700=1042.461,393.028,-130.708,173.826,43.673,158.603
C04701=1042.451,392.781,-130.665,173.818,43.667,158.601
C04702=1042.442,392.536,-130.621,173.810,43.662,158.599
C04703=1042.434,392.290,-130.578,173.802,43.657,158.597
C04704=1042.426,392.059,-130.539,173.795,43.652,158.595
C04705=1042.417,391.829,-130.498,173.787,43.647,158.594
C04706=1042.409,391.599,-130.458,173.780,43.642,158.592
C04707=1042.401,391.369,-130.418,173.772,43.637,158.590
C04708=1042.393,391.139,-130.378,173.766,43.632,158.588
C04709=1042.385,390.909,-130.339,173.758,43.626,158.586
C04710=1042.376,390.679,-130.298,173.751,43.622,158.584
C04711=1042.368,390.449,-130.258,173.744,43.617,158.582
C04712=1042.359,390.203,-130.216,173.736,43.612,158.580
C04713=1042.351,389.956,-130.173,173.728,43.606,158.578
C04714=1042.341,389.711,-130.131,173.720,43.601,158.576
C04715=1042.333,389.464,-130.088,173.713,43.596,158.575
C04716=1042.324,389.218,-130.046,173.705,43.591,158.573
C04717=1042.315,388.972,-130.003,173.697,43.586,158.571
C04718=1042.306,388.726,-129.961,173.690,43.580,158.569
C04719=1042.298,388.480,-129.918,173.682,43.576,158.567
C04720=1042.289,388.234,-129.876,173.674,43.570,158.565
C04721=1042.281,387.987,-129.834,173.667,43.565,158.563
C04722=1042.272,387.741,-129.792,173.659,43.560,158.561
C04723=1042.262,387.495,-129.749,173.652,43.555,158.559
C04724=1042.253,387.249,-129.708,173.644,43.550,158.557
C04725=1042.245,387.002,-129.665,173.637,43.545,158.555
C04726=1042.236,386.756,-129.624,173.629,43.540,158.554
C04727=1042.227,386.510,-129.581,173.621,43.535,158.552
C04728=1042.219,386.263,-129.539,173.614,43.530,158.550
C04729=1042.210,386.017,-129.497,173.606,43.525,158.548
C04730=1042.201,385.771,-129.455,173.599,43.520,158.546
C04731=1042.193,385.525,-129.414,173.591,43.515,158.544
C04732=1042.184,385.278,-129.372,173.584,43.510,158.542
C04733=1042.176,385.032,-129.330,173.577,43.506,158.541
C04734=1042.167,384.785,-129.288,173.569,43.501,158.539
C04735=1042.157,384.540,-129.246,173.562,43.495,158.537
C04736=1042.150,384.293,-129.205,173.555,43.491,158.535
C04737=1042.141,384.047,-129.163,173.547,43.486,158.533
C04738=1042.132,383.800,-129.121,173.540,43.481,158.531
C04739=1042.124,383.555,-129.080,173.533,43.476,158.530
C04740=1042.116,383.308,-129.038,173.525,43.471,158.528
C04741=1042.107,383.062,-128.996,173.518,43.466,158.526
C04742=1042.098,382.815,-128.954,173.511,43.462,158.524
C04743=1042.090,382.569,-128.914,173.503,43.457,158.522
C04744=1042.081,382.323,-128.872,173.497,43.452,158.521
C04745=1042.073,382.077,-128.830,173.490,43.448,158.519
C04746=1042.064,381.830,-128.788,173.483,43.443,158.517
C04747=1042.056,381.583,-128.747,173.475,43.438,158.515
C04748=1042.047,381.338,-128.706,173.468,43.433,158.514
C04749=1042.039,381.091,-128.664,173.461,43.429,158.512
C04750=1042.031,380.845,-128.623,173.454,43.424,158.510
C04751=1042.022,380.598,-128.581,173.446,43.419,158.508
C04752=1042.014,380.352,-128.541,173.440,43.415,158.507
C04753=1042.005,380.106,-128.499,173.433,43.410,158.505
C04754=1041.998,379.859,-128.458,173.426,43.405,158.503
C04755=1041.989,379.613,-128.416,173.419,43.401,158.501
C04756=1041.981,379.367,-128.375,173.411,43.396,158.500
C04757=1041.972,379.120,-128.334,173.405,43.391,158.498
C04758=1041.964,378.874,-128.293,173.398,43.386,158.496
C04759=1041.956,378.628,-128.252,173.391,43.382,158.495
C04760=1041.947,378.381,-128.211,173.384,43.378,158.493
C04761=1041.939,378.134,-128.171,173.378,43.373,158.491
C04762=1041.931,377.887,-128.130,173.370,43.368,158.490
C04763=1041.922,377.642,-128.088,173.363,43.364,158.488
C04764=1041.910,377.272,-128.028,173.353,43.357,158.485
C04765=1041.897,376.901,-127.966,173.343,43.350,158.483
C04766=1041.885,376.531,-127.905,173.333,43.344,158.480
C04767=1041.872,376.162,-127.845,173.323,43.337,158.478
C04768=1041.864,375.915,-127.804,173.316,43.333,158.476
C04769=1041.855,375.668,-127.763,173.309,43.328,158.475
C04770=1041.847,375.422,-127.722,173.301,43.324,158.473
C04771=1041.839,375.176,-127.682,173.295,43.319,158.471
C04772=1041.831,374.929,-127.641,173.288,43.315,158.470
C04773=1041.823,374.682,-127.600,173.282,43.311,158.468
C04774=1041.814,374.436,-127.561,173.275,43.306,158.467
C04775=1041.806,374.190,-127.520,173.268,43.302,158.465
C04776=1041.798,373.943,-127.480,173.262,43.298,158.464
C04777=1041.790,373.697,-127.439,173.255,43.294,158.462
C04778=1041.782,373.449,-127.399,173.248,43.289,158.460
C04779=1041.774,373.203,-127.358,173.242,43.285,158.459
C04780=1041.765,372.957,-127.318,173.235,43.281,158.457
C04781=1041.757,372.710,-127.278,173.229,43.276,158.456
C04782=1041.749,372.464,-127.237,173.222,43.272,158.454
C04783=1041.742,372.217,-127.197,173.215,43.268,158.452
C04784=1041.734,371.971,-127.157,173.209,43.264,158.451
C04785=1041.726,371.724,-127.117,173.202,43.259,158.449
C04786=1041.717,371.478,-127.077,173.196,43.255,158.448
C04787=1041.709,371.231,-127.037,173.189,43.251,158.446
C04788=1041.701,370.985,-126.996,173.184,43.247,158.445
C04789=1041.693,370.737,-126.956,173.177,43.243,158.443
C04790=1041.685,370.490,-126.916,173.171,43.238,158.442
C04791=1041.676,370.244,-126.876,173.164,43.234,158.440
C04792=1041.669,369.997,-126.836,173.158,43.230,158.439
C04793=1041.660,369.751,-126.797,173.151,43.226,158.437
C04794=1041.653,369.504,-126.757,173.145,43.222,158.436
C04795=1041.644,369.257,-126.718,173.138,43.218,158.434
C04796=1041.636,369.010,-126.678,173.132,43.214,158.433
C04797=1041.628,368.764,-126.638,173.125,43.210,158.431
C04798=1041.620,368.517,-126.598,173.119,43.206,158.430
C04799=1041.611,368.271,-126.558,173.113,43.202,158.428
C04800=1041.604,368.024,-126.518,173.107,43.198,158.427
C04801=1041.595,367.777,-126.479,173.100,43.194,158.425
C04802=1041.588,367.531,-126.440,173.094,43.190,158.424
C04803=1041.580,367.285,-126.400,173.088,43.186,158.422
C04804=1041.572,367.038,-126.360,173.081,43.182,158.421
C04805=1041.564,366.790,-126.322,173.076,43.178,158.419
C04806=1041.556,366.543,-126.282,173.069,43.174,158.418
C04807=1041.548,366.297,-126.243,173.063,43.170,158.417
C04808=1041.540,366.050,-126.203,173.056,43.166,158.415
C04809=1041.532,365.804,-126.164,173.050,43.162,158.414
C04810=1041.524,365.557,-126.124,173.044,43.158,158.412
C04811=1041.516,365.310,-126.085,173.038,43.154,158.411
C04812=1041.508,365.063,-126.045,173.032,43.150,158.409
C04813=1041.500,364.816,-126.006,173.026,43.146,158.408
C04814=1041.493,364.570,-125.966,173.019,43.142,158.406
C04815=1041.485,364.323,-125.928,173.013,43.138,158.405
C04816=1041.476,364.076,-125.888,173.008,43.135,158.404
C04817=1041.469,363.830,-125.850,173.001,43.131,158.402
C04818=1041.461,363.583,-125.810,172.995,43.127,158.401
C04819=1041.453,363.336,-125.770,172.990,43.123,158.400
C04820=1041.442,362.986,-125.715,172.981,43.118,158.398
C04821=1041.432,362.636,-125.660,172.973,43.112,158.396
C04822=1041.420,362.286,-125.604,172.964,43.107,158.394
C04823=1041.409,361.936,-125.549,172.955,43.102,158.392
C04824=1041.401,361.689,-125.511,172.949,43.098,158.390
C04825=1041.393,361.442,-125.471,172.943,43.094,158.389
C04826=1041.386,361.195,-125.433,172.938,43.090,158.388
C04827=1041.378,360.948,-125.394,172.931,43.087,158.386
C04828=1041.370,360.702,-125.355,172.925,43.083,158.385
C04829=1041.362,360.455,-125.316,172.920,43.079,158.383
C04830=1041.354,360.207,-125.277,172.914,43.075,158.382
C04831=1041.347,359.961,-125.239,172.907,43.072,158.381
C04832=1041.339,359.714,-125.200,172.901,43.068,158.379
C04833=1041.331,359.467,-125.162,172.896,43.065,158.378
C04834=1041.323,359.220,-125.123,172.890,43.061,158.377
C04835=1041.315,358.973,-125.085,172.885,43.057,158.376
C04836=1041.308,358.727,-125.045,172.878,43.054,158.374
C04837=1041.300,358.480,-125.007,172.872,43.050,158.373
C04838=1041.292,358.233,-124.968,172.867,43.047,158.372
C04839=1041.284,357.986,-124.930,172.861,43.043,158.370
C04840=1041.277,357.738,-124.892,172.855,43.039,158.369
C04841=1041.269,357.492,-124.854,172.850,43.036,158.368
C04842=1041.261,357.245,-124.815,172.843,43.033,158.366
C04843=1041.253,356.998,-124.777,172.838,43.029,158.365
C04844=1041.246,356.751,-124.738,172.832,43.025,158.364
C04845=1041.238,356.504,-124.700,172.826,43.022,158.363
C04846=1041.231,356.258,-124.662,172.821,43.018,158.361
C04847=1041.223,356.010,-124.624,172.815,43.015,158.360
C04848=1041.215,355.764,-124.586,172.810,43.011,158.359
C04849=1041.206,355.516,-124.547,172.803,43.008,158.357
C04850=1041.199,355.269,-124.510,172.797,43.004,158.356
C04851=1041.192,355.023,-124.472,172.792,43.001,158.355
C04852=1041.184,354.776,-124.433,172.786,42.997,158.354
C04853=1041.176,354.528,-124.396,172.781,42.994,158.352
C04854=1041.169,354.282,-124.357,172.775,42.991,158.351
C04855=1041.161,354.035,-124.319,172.770,42.987,158.350
C04856=1041.153,353.788,-124.281,172.764,42.984,158.349
C04857=1041.146,353.541,-124.243,172.759,42.980,158.347
C04858=1041.138,353.293,-124.205,172.753,42.977,158.346
C04859=1041.130,353.047,-124.167,172.748,42.973,158.345
C04860=1041.123,352.800,-124.129,172.742,42.970,158.344
C04861=1041.115,352.553,-124.092,172.737,42.966,158.343
C04862=1041.107,352.306,-124.054,172.731,42.963,158.341
C04863=1041.100,352.058,-124.016,172.725,42.960,158.340
C04864=1041.092,351.812,-123.978,172.720,42.957,158.339
C04865=1041.085,351.565,-123.940,172.715,42.953,158.338
C04866=1041.078,351.318,-123.903,172.709,42.950,158.337
C04867=1041.070,351.070,-123.864,172.704,42.946,158.335
C04868=1041.062,350.823,-123.827,172.698,42.943,158.334
C04869=1041.055,350.576,-123.789,172.693,42.940,158.333
C04870=1041.047,350.329,-123.752,172.687,42.937,158.332
C04871=1041.040,350.083,-123.714,172.682,42.933,158.331
C04872=1041.032,349.836,-123.676,172.676,42.930,158.329
C04873=1041.024,349.588,-123.639,172.671,42.927,158.328
C04874=1041.016,349.341,-123.602,172.665,42.924,158.327
C04875=1041.009,349.094,-123.564,172.660,42.920,158.326
C04876=1040.999,348.750,-123.512,172.652,42.916,158.324
C04877=1040.988,348.405,-123.460,172.645,42.911,158.323
C04878=1040.978,348.062,-123.407,172.637,42.907,158.321
C04879=1040.967,347.718,-123.356,172.630,42.903,158.319
C04880=1040.960,347.470,-123.319,172.624,42.899,158.318
C04881=1040.953,347.223,-123.281,172.619,42.896,158.317
C04882=1040.945,346.976,-123.244,172.614,42.893,158.316
C04883=1040.937,346.729,-123.207,172.608,42.890,158.315
C04884=1040.930,346.482,-123.169,172.603,42.886,158.314
C04885=1040.922,346.235,-123.133,172.597,42.884,158.312
C04886=1040.915,345.988,-123.096,172.592,42.881,158.311
C04887=1040.907,345.741,-123.059,172.588,42.877,158.310
C04888=1040.900,345.494,-123.021,172.582,42.874,158.309
C04889=1040.893,345.247,-122.984,172.577,42.871,158.308
C04890=1040.885,344.999,-122.947,172.571,42.868,158.307
C04891=1040.878,344.752,-122.910,172.566,42.865,158.306
C04892=1040.870,344.505,-122.873,172.561,42.862,158.305
C04893=1040.863,344.257,-122.836,172.555,42.859,158.303
C04894=1040.855,344.011,-122.799,172.551,42.856,158.302
C04895=1040.848,343.763,-122.762,172.546,42.853,158.301
C04896=1040.841,343.516,-122.725,172.540,42.849,158.300
C04897=1040.833,343.269,-122.688,172.535,42.846,158.299
C04898=1040.826,343.022,-122.651,172.530,42.843,158.298
C04899=1040.818,342.775,-122.615,172.525,42.840,158.297
C04900=1040.812,342.527,-122.578,172.520,42.838,158.296
C04901=1040.804,342.280,-122.541,172.515,42.834,158.295
C04902=1040.797,342.033,-122.504,172.509,42.831,158.294
C04903=1040.789,341.786,-122.467,172.504,42.828,158.292
C04904=1040.782,341.539,-122.431,172.500,42.825,158.291
C04905=1040.775,341.291,-122.394,172.494,42.822,158.290
C04906=1040.767,341.044,-122.357,172.489,42.819,158.289
C04907=1040.759,340.797,-122.321,172.484,42.817,158.288
C04908=1040.752,340.549,-122.284,172.478,42.814,158.287
C04909=1040.744,340.302,-122.248,172.474,42.811,158.286
C04910=1040.737,340.056,-122.212,172.469,42.808,158.285
C04911=1040.730,339.808,-122.175,172.464,42.805,158.284
C04912=1040.722,339.560,-122.139,172.458,42.802,158.283
C04913=1040.715,339.313,-122.102,172.454,42.799,158.282
C04914=1040.708,339.066,-122.067,172.449,42.796,158.281
C04915=1040.700,338.819,-122.029,172.443,42.793,158.280
C04916=1040.693,338.572,-121.993,172.438,42.790,158.279
C04917=1040.685,338.324,-121.957,172.434,42.788,158.278
C04918=1040.678,338.078,-121.921,172.429,42.785,158.277
C04919=1040.671,337.830,-121.884,172.423,42.782,158.276
C04920=1040.663,337.582,-121.848,172.419,42.779,158.275
C04921=1040.656,337.336,-121.812,172.414,42.776,158.274
C04922=1040.649,337.088,-121.775,172.409,42.773,158.273
C04923=1040.642,336.840,-121.739,172.405,42.771,158.272
C04924=1040.635,336.594,-121.703,172.399,42.768,158.271
C04925=1040.627,336.346,-121.667,172.394,42.765,158.270
C04926=1040.621,336.099,-121.630,172.390,42.762,158.269
C04927=1040.613,335.852,-121.594,172.384,42.759,158.267
C04928=1040.605,335.604,-121.558,172.379,42.757,158.267
C04929=1040.598,335.357,-121.522,172.375,42.753,158.266
C04930=1040.591,335.109,-121.487,172.370,42.751,158.264
C04931=1040.584,334.863,-121.451,172.365,42.748,158.264
C04932=1040.573,334.514,-121.399,172.358,42.744,158.262
C04933=1040.563,334.166,-121.349,172.351,42.740,158.261
C04934=1040.553,333.819,-121.299,172.344,42.736,158.259
C04935=1040.543,333.471,-121.249,172.338,42.733,158.258
C04936=1040.535,333.224,-121.213,172.333,42.730,158.257
C04937=1040.528,332.977,-121.177,172.328,42.727,158.256
C04938=1040.520,332.729,-121.141,172.323,42.725,158.255
C04939=1040.513,332.482,-121.105,172.318,42.722,158.254
C04940=1040.506,332.234,-121.070,172.314,42.719,158.253
C04941=1040.499,331.987,-121.034,172.309,42.717,158.252
C04942=1040.491,331.740,-120.998,172.305,42.714,158.251
C04943=1040.484,331.493,-120.963,172.299,42.711,158.250
C04944=1040.477,331.246,-120.927,172.294,42.709,158.249
C04945=1040.470,330.998,-120.891,172.290,42.706,158.248
C04946=1040.463,330.751,-120.855,172.285,42.703,158.247
C04947=1040.456,330.503,-120.820,172.281,42.701,158.246
C04948=1040.449,330.256,-120.785,172.276,42.698,158.245
C04949=1040.441,330.008,-120.749,172.272,42.695,158.245
C04950=1040.434,329.761,-120.713,172.266,42.693,158.244
C04951=1040.427,329.514,-120.678,172.262,42.690,158.243
C04952=1040.420,329.266,-120.642,172.257,42.688,158.242
C04953=1040.413,329.019,-120.607,172.253,42.685,158.241
C04954=1040.406,328.772,-120.571,172.248,42.682,158.240
C04955=1040.398,328.524,-120.536,172.243,42.680,158.239
C04956=1040.391,328.277,-120.501,172.239,42.678,158.238
C04957=1040.384,328.029,-120.466,172.234,42.675,158.237
C04958=1040.376,327.782,-120.431,172.229,42.672,158.236
C04959=1040.370,327.534,-120.396,172.224,42.670,158.235
C04960=1040.361,327.287,-120.360,172.220,42.667,158.234
C04961=1040.354,327.040,-120.325,172.215,42.665,158.233
C04962=1040.347,326.793,-120.291,172.211,42.662,158.233
C04963=1040.339,326.545,-120.255,172.206,42.660,158.232
C04964=1040.333,326.297,-120.220,172.202,42.658,158.231
C04965=1040.325,326.050,-120.185,172.197,42.655,158.230
C04966=1040.318,325.802,-120.150,172.193,42.653,158.229
C04967=1040.310,325.555,-120.115,172.188,42.650,158.228
C04968=1040.304,325.308,-120.080,172.184,42.648,158.227
C04969=1040.295,325.060,-120.045,172.179,42.646,158.226
C04970=1040.289,324.813,-120.010,172.175,42.643,158.226
C04971=1040.281,324.566,-119.976,172.170,42.641,158.225
C04972=1040.274,324.318,-119.941,172.165,42.638,158.224
C04973=1040.267,324.070,-119.906,172.160,42.636,158.223
C04974=1040.260,323.823,-119.871,172.156,42.633,158.222
C04975=1040.253,323.575,-119.836,172.151,42.631,158.221
C04976=1040.246,323.328,-119.802,172.147,42.629,158.220
C04977=1040.239,323.081,-119.766,172.142,42.626,158.219
C04978=1040.231,322.833,-119.732,172.138,42.624,158.218
C04979=1040.224,322.585,-119.697,172.134,42.621,158.218
C04980=1040.217,322.338,-119.663,172.129,42.619,158.217
C04981=1040.210,322.091,-119.627,172.125,42.616,158.216
C04982=1040.202,321.844,-119.593,172.120,42.614,158.215
C04983=1040.196,321.596,-119.558,172.116,42.611,158.214
C04984=1040.188,321.348,-119.524,172.111,42.610,158.213
C04985=1040.181,321.100,-119.488,172.107,42.607,158.212
C04986=1040.174,320.853,-119.455,172.103,42.605,158.212
C04987=1040.167,320.605,-119.419,172.098,42.602,158.211
C04988=1040.157,320.253,-119.370,172.091,42.599,158.209
C04989=1040.147,319.900,-119.321,172.086,42.595,158.208
C04990=1040.137,319.548,-119.272,172.079,42.592,158.207
C04991=1040.127,319.195,-119.223,172.073,42.589,158.206
C04992=1040.120,318.948,-119.188,172.069,42.587,158.205
C04993=1040.113,318.700,-119.153,172.064,42.584,158.204
C04994=1040.106,318.453,-119.119,172.060,42.582,158.203
C04995=1040.099,318.205,-119.084,172.056,42.579,158.202
C04996=1040.092,317.958,-119.050,172.051,42.578,158.202
C04997=1040.085,317.710,-119.016,172.047,42.575,158.201
C04998=1040.078,317.463,-118.981,172.043,42.573,158.200
C04999=1040.071,317.216,-118.948,172.038,42.570,158.199
C05000=1040.065,316.968,-118.913,172.034,42.568,158.198
C05001=1040.057,316.721,-118.879,172.030,42.566,158.198
C05002=1040.051,316.473,-118.844,172.026,42.563,158.197
C05003=1040.043,316.226,-118.810,172.021,42.561,158.196
C05004=1040.037,315.978,-118.775,172.017,42.559,158.195
C05005=1040.029,315.731,-118.741,172.013,42.556,158.194
C05006=1040.023,315.483,-118.706,172.008,42.555,158.193
C05007=1040.016,315.235,-118.673,172.004,42.552,158.193
C05008=1040.010,314.988,-118.638,172.000,42.550,158.192
C05009=1040.002,314.741,-118.604,171.996,42.548,158.191
C05010=1039.996,314.493,-118.570,171.991,42.545,158.190
C05011=1039.989,314.245,-118.536,171.987,42.543,158.189
C05012=1039.981,313.998,-118.501,171.983,42.541,158.189
C05013=1039.975,313.750,-118.467,171.979,42.538,158.188
C05014=1039.968,313.503,-118.433,171.974,42.537,158.187
C05015=1039.962,313.255,-118.399,171.970,42.534,158.186
C05016=1039.954,313.007,-118.365,171.966,42.532,158.185
C05017=1039.948,312.759,-118.331,171.962,42.530,158.185
C05018=1039.941,312.513,-118.297,171.957,42.527,158.184
C05019=1039.935,312.265,-118.262,171.954,42.525,158.183
C05020=1039.927,312.017,-118.228,171.950,42.523,158.182
C05021=1039.920,311.770,-118.194,171.946,42.521,158.181
C05022=1039.913,311.522,-118.161,171.941,42.519,158.181
C05023=1039.906,311.275,-118.128,171.937,42.517,158.180
C05024=1039.899,311.027,-118.095,171.933,42.515,158.179
C05025=1039.892,310.779,-118.061,171.929,42.513,158.178
C05026=1039.884,310.532,-118.027,171.924,42.511,158.178
C05027=1039.877,310.284,-117.993,171.920,42.508,158.177
C05028=1039.870,310.036,-117.959,171.916,42.506,158.176
C05029=1039.864,309.789,-117.927,171.913,42.504,158.175
C05030=1039.856,309.541,-117.893,171.908,42.503,158.175
C05031=1039.849,309.294,-117.860,171.904,42.500,158.174
C05032=1039.841,309.046,-117.826,171.900,42.498,158.173
C05033=1039.835,308.798,-117.793,171.896,42.496,158.172
C05034=1039.828,308.551,-117.759,171.892,42.494,158.172
C05035=1039.821,308.303,-117.725,171.887,42.492,158.171
C05036=1039.814,308.056,-117.692,171.883,42.490,158.170
C05037=1039.806,307.808,-117.659,171.879,42.488,158.169
C05038=1039.799,307.560,-117.626,171.876,42.486,158.169
C05039=1039.793,307.313,-117.592,171.872,42.484,158.168
C05040=1039.786,307.065,-117.559,171.867,42.482,158.167
C05041=1039.779,306.817,-117.525,171.863,42.480,158.166
C05042=1039.772,306.570,-117.492,171.859,42.478,158.166
C05043=1039.764,306.323,-117.459,171.855,42.476,158.165
C05044=1039.755,305.974,-117.412,171.849,42.473,158.164
C05045=1039.745,305.627,-117.366,171.844,42.470,158.163
C05046=1039.735,305.279,-117.318,171.839,42.468,158.162
C05047=1039.726,304.931,-117.272,171.832,42.465,158.161
C05048=1039.719,304.683,-117.239,171.829,42.463,158.160
C05049=1039.711,304.436,-117.206,171.825,42.461,158.159
C05050=1039.704,304.188,-117.173,171.821,42.459,158.159
C05051=1039.698,303.941,-117.139,171.817,42.457,158.158
C05052=1039.691,303.693,-117.106,171.813,42.455,158.157
C05053=1039.684,303.445,-117.073,171.808,42.453,158.156
C05054=1039.677,303.198,-117.040,171.804,42.451,158.156
C05055=1039.670,302.950,-117.007,171.801,42.449,158.155
C05056=1039.663,302.703,-116.974,171.797,42.447,158.154
C05057=1039.656,302.454,-116.941,171.793,42.445,158.154
C05058=1039.650,302.207,-116.908,171.789,42.443,158.153
C05059=1039.643,301.959,-116.874,171.785,42.441,158.152
C05060=1039.636,301.712,-116.842,171.781,42.439,158.152
C05061=1039.630,301.464,-116.809,171.778,42.437,158.151
C05062=1039.623,301.216,-116.776,171.774,42.435,158.150
C05063=1039.616,300.969,-116.743,171.770,42.433,158.149
C05064=1039.608,300.721,-116.710,171.766,42.431,158.149
C05065=1039.602,300.473,-116.677,171.761,42.430,158.148
C05066=1039.595,300.225,-116.644,171.757,42.428,158.147
C05067=1039.589,299.978,-116.611,171.754,42.426,158.147
C05068=1039.582,299.730,-116.578,171.750,42.424,158.146
C05069=1039.575,299.483,-116.546,171.746,42.422,158.145
C05070=1039.568,299.235,-116.513,171.742,42.420,158.145
C05071=1039.561,298.987,-116.480,171.738,42.418,158.144
C05072=1039.555,298.739,-116.447,171.734,42.416,158.143
C05073=1039.548,298.492,-116.415,171.731,42.414,158.142
C05074=1039.541,298.244,-116.381,171.727,42.412,158.142
C05075=1039.535,297.997,-116.348,171.723,42.410,158.141
C05076=1039.528,297.749,-116.315,171.719,42.408,158.140
C05077=1039.521,297.501,-116.282,171.715,42.406,158.140
C05078=1039.514,297.253,-116.250,171.712,42.405,158.139
C05079=1039.508,297.006,-116.217,171.708,42.403,158.138
C05080=1039.501,296.757,-116.184,171.704,42.401,158.138
C05081=1039.495,296.510,-116.152,171.700,42.399,158.137
C05082=1039.488,296.263,-116.119,171.696,42.397,158.136
C05083=1039.481,296.014,-116.086,171.693,42.395,158.136
C05084=1039.475,295.767,-116.054,171.689,42.393,158.135
C05085=1039.468,295.519,-116.021,171.686,42.391,158.134
C05086=1039.461,295.272,-115.989,171.682,42.389,158.133
C05087=1039.455,295.023,-115.956,171.679,42.388,158.133
C05088=1039.448,294.776,-115.924,171.675,42.386,158.132
C05089=1039.442,294.528,-115.891,171.671,42.384,158.132
C05090=1039.434,294.280,-115.859,171.667,42.382,158.131
C05091=1039.427,294.032,-115.827,171.663,42.381,158.130
C05092=1039.421,293.785,-115.795,171.660,42.379,158.130
C05093=1039.413,293.537,-115.762,171.656,42.377,158.129
C05094=1039.407,293.289,-115.729,171.652,42.375,158.128
C05095=1039.400,293.041,-115.698,171.648,42.373,158.128
C05096=1039.393,292.794,-115.666,171.644,42.371,158.127
C05097=1039.386,292.546,-115.633,171.641,42.370,158.126
C05098=1039.380,292.298,-115.601,171.637,42.368,158.126
C05099=1039.373,292.050,-115.569,171.633,42.366,158.125
C05100=1039.364,291.719,-115.526,171.628,42.364,158.124
C05101=1039.355,291.388,-115.483,171.623,42.362,158.123
C05102=1039.345,291.057,-115.440,171.618,42.359,158.123
C05103=1039.336,290.725,-115.397,171.613,42.357,158.122
C05104=1039.330,290.477,-115.365,171.610,42.356,158.121
C05105=1039.322,290.230,-115.333,171.607,42.354,158.120
C05106=1039.316,289.982,-115.301,171.603,42.352,158.120
C05107=1039.309,289.735,-115.269,171.599,42.350,158.119
C05108=1039.302,289.486,-115.237,171.596,42.348,158.118
C05109=1039.296,289.238,-115.205,171.592,42.347,158.118
C05110=1039.289,288.991,-115.173,171.588,42.345,158.117
C05111=1039.282,288.743,-115.142,171.585,42.344,158.117
C05112=1039.275,288.495,-115.110,171.581,42.342,158.116
C05113=1039.269,288.247,-115.078,171.577,42.340,158.115
C05114=1039.262,287.999,-115.045,171.573,42.338,158.115
C05115=1039.255,287.751,-115.014,171.571,42.337,158.114
C05116=1039.248,287.503,-114.982,171.567,42.335,158.114
C05117=1039.241,287.256,-114.950,171.563,42.333,158.113
C05118=1039.235,287.008,-114.919,171.559,42.331,158.112
C05119=1039.229,286.760,-114.887,171.556,42.330,158.112
C05120=1039.222,286.512,-114.855,171.552,42.328,158.111
C05121=1039.214,286.264,-114.823,171.548,42.327,158.111
C05122=1039.207,286.016,-114.791,171.545,42.325,158.110
C05123=1039.201,285.768,-114.760,171.542,42.323,158.109
C05124=1039.194,285.520,-114.728,171.538,42.322,158.109
C05125=1039.187,285.272,-114.697,171.534,42.320,158.108
C05126=1039.181,285.025,-114.665,171.531,42.319,158.108
C05127=1039.174,284.777,-114.633,171.527,42.317,158.107
C05128=1039.167,284.529,-114.602,171.523,42.315,158.106
C05129=1039.160,284.282,-114.570,171.520,42.314,158.106
C05130=1039.153,284.034,-114.539,171.517,42.312,158.105
C05131=1039.147,283.786,-114.508,171.513,42.310,158.105
C05132=1039.140,283.538,-114.476,171.510,42.309,158.104
C05133=1039.133,283.289,-114.444,171.506,42.307,158.103
C05134=1039.126,283.041,-114.413,171.502,42.306,158.103
C05135=1039.119,282.793,-114.382,171.500,42.304,158.102
C05136=1039.112,282.545,-114.350,171.496,42.302,158.102
C05137=1039.106,282.298,-114.319,171.492,42.301,158.101
C05138=1039.099,282.050,-114.287,171.489,42.299,158.100
C05139=1039.092,281.802,-114.256,171.485,42.297,158.100
C05140=1039.086,281.554,-114.224,171.482,42.296,158.099
C05141=1039.079,281.306,-114.193,171.479,42.294,158.099
C05142=1039.072,281.058,-114.161,171.475,42.293,158.098
C05143=1039.065,280.810,-114.130,171.471,42.291,158.097
C05144=1039.059,280.563,-114.099,171.468,42.290,158.097
C05145=1039.052,280.315,-114.068,171.465,42.288,158.096
C05146=1039.046,280.067,-114.037,171.461,42.286,158.096
C05147=1039.039,279.819,-114.006,171.458,42.285,158.095
C05148=1039.032,279.571,-113.975,171.454,42.283,158.094
C05149=1039.025,279.323,-113.943,171.451,42.281,158.094
C05150=1039.018,279.075,-113.912,171.447,42.280,158.093
C05151=1039.012,278.827,-113.880,171.444,42.279,158.093
C05152=1039.005,278.579,-113.850,171.440,42.277,158.092
C05153=1038.999,278.331,-113.818,171.437,42.275,158.092
C05154=1038.992,278.083,-113.787,171.434,42.274,158.091
C05155=1038.985,277.835,-113.755,171.430,42.272,158.091
C05156=1038.976,277.516,-113.715,171.426,42.270,158.090
C05157=1038.968,277.196,-113.676,171.422,42.269,158.089
C05158=1038.959,276.877,-113.636,171.418,42.267,158.088
C05159=1038.950,276.558,-113.596,171.413,42.265,158.088
C05160=1038.944,276.310,-113.565,171.409,42.263,158.087
C05161=1038.937,276.062,-113.534,171.407,42.261,158.087
C05162=1038.930,275.814,-113.503,171.403,42.260,158.086
C05163=1038.923,275.566,-113.472,171.399,42.258,158.085
C05164=1038.917,275.318,-113.442,171.396,42.257,158.085
C05165=1038.910,275.071,-113.411,171.393,42.256,158.084
C05166=1038.903,274.822,-113.380,171.389,42.254,158.084
C05167=1038.897,274.574,-113.349,171.386,42.252,158.083
C05168=1038.890,274.326,-113.318,171.383,42.251,158.083
C05169=1038.883,274.078,-113.287,171.379,42.249,158.082
C05170=1038.877,273.830,-113.257,171.376,42.248,158.082
C05171=1038.870,273.582,-113.225,171.372,42.247,158.081
C05172=1038.863,273.334,-113.195,171.370,42.245,158.081
C05173=1038.856,273.086,-113.164,171.366,42.244,158.080
C05174=1038.849,272.838,-113.134,171.362,42.242,158.079
C05175=1038.843,272.590,-113.103,171.360,42.241,158.079
C05176=1038.837,272.342,-113.072,171.356,42.239,158.078
C05177=1038.829,272.094,-113.042,171.353,42.238,158.078
C05178=1038.823,271.846,-113.011,171.350,42.236,158.077
C05179=1038.817,271.598,-112.980,171.346,42.234,158.077
C05180=1038.810,271.350,-112.950,171.342,42.233,158.076
C05181=1038.803,271.102,-112.919,171.340,42.231,158.076
C05182=1038.796,270.854,-112.888,171.336,42.230,158.075
C05183=1038.789,270.606,-112.858,171.333,42.229,158.075
C05184=1038.783,270.358,-112.828,171.330,42.227,158.074
C05185=1038.776,270.110,-112.796,171.326,42.226,158.073
C05186=1038.769,269.862,-112.766,171.324,42.224,158.073
C05187=1038.763,269.613,-112.736,171.320,42.223,158.072
C05188=1038.756,269.366,-112.706,171.317,42.222,158.072
C05189=1038.750,269.117,-112.675,171.314,42.220,158.071
C05190=1038.742,268.870,-112.644,171.310,42.219,158.071
C05191=1038.736,268.622,-112.614,171.307,42.217,158.070
C05192=1038.729,268.374,-112.584,171.304,42.216,158.070
C05193=1038.722,268.126,-112.554,171.301,42.215,158.069
C05194=1038.716,267.877,-112.523,171.297,42.214,158.069
C05195=1038.709,267.630,-112.493,171.295,42.212,158.068
C05196=1038.703,267.381,-112.462,171.291,42.211,158.068
C05197=1038.695,267.133,-112.432,171.288,42.209,158.067
C05198=1038.690,266.885,-112.402,171.285,42.208,158.067
C05199=1038.682,266.637,-112.372,171.281,42.206,158.066
C05200=1038.675,266.389,-112.341,171.278,42.205,158.066
C05201=1038.668,266.142,-112.311,171.275,42.203,158.065
C05202=1038.662,265.893,-112.281,171.272,42.202,158.065
C05203=1038.655,265.644,-112.251,171.269,42.200,158.064
C05204=1038.649,265.397,-112.221,171.265,42.200,158.064
C05205=1038.642,265.148,-112.191,171.263,42.198,158.063
C05206=1038.635,264.900,-112.161,171.259,42.197,158.063
C05207=1038.629,264.653,-112.131,171.256,42.195,158.062
C05208=1038.622,264.404,-112.100,171.253,42.194,158.062
C05209=1038.616,264.157,-112.070,171.250,42.192,158.061
C05210=1038.608,263.908,-112.040,171.247,42.191,158.061
C05211=1038.602,263.660,-112.009,171.243,42.190,158.060
C05212=1038.593,263.345,-111.972,171.239,42.188,158.059
C05213=1038.585,263.031,-111.933,171.236,42.186,158.059
C05214=1038.576,262.716,-111.896,171.232,42.185,158.058
C05215=1038.568,262.401,-111.858,171.227,42.183,158.058
C05216=1038.562,262.153,-111.828,171.225,42.181,158.057
C05217=1038.555,261.905,-111.798,171.221,42.180,158.057
C05218=1038.548,261.658,-111.768,171.219,42.179,158.056
C05219=1038.541,261.409,-111.739,171.215,42.178,158.056
C05220=1038.534,261.160,-111.708,171.212,42.176,158.055
C05221=1038.527,260.913,-111.679,171.209,42.175,158.055
C05222=1038.521,260.664,-111.649,171.206,42.174,158.054
C05223=1038.514,260.417,-111.619,171.203,42.172,158.054
C05224=1038.507,260.168,-111.589,171.199,42.172,158.053
C05225=1038.500,259.920,-111.560,171.197,42.170,158.053
C05226=1038.493,259.672,-111.530,171.193,42.169,158.052
C05227=1038.487,259.423,-111.501,171.191,42.168,158.052
C05228=1038.480,259.176,-111.471,171.187,42.166,158.051
C05229=1038.473,258.927,-111.442,171.184,42.165,158.051
C05230=1038.466,258.680,-111.412,171.181,42.164,158.050
C05231=1038.459,258.431,-111.383,171.178,42.162,158.050
C05232=1038.452,258.183,-111.353,171.175,42.161,158.049
C05233=1038.445,257.935,-111.323,171.172,42.160,158.049
C05234=1038.439,257.686,-111.294,171.169,42.159,158.048
C05235=1038.432,257.438,-111.265,171.166,42.157,158.048
C05236=1038.425,257.190,-111.235,171.163,42.156,158.048
C05237=1038.419,256.942,-111.206,171.160,42.155,158.047
C05238=1038.412,256.694,-111.175,171.157,42.153,158.047
C05239=1038.405,256.445,-111.146,171.154,42.152,158.046
C05240=1038.398,256.198,-111.117,171.151,42.151,158.046
C05241=1038.391,255.949,-111.088,171.148,42.149,158.045
C05242=1038.384,255.701,-111.058,171.145,42.149,158.045
C05243=1038.378,255.453,-111.029,171.142,42.147,158.044
C05244=1038.371,255.204,-110.999,171.138,42.146,158.044
C05245=1038.365,254.957,-110.970,171.136,42.145,158.043
C05246=1038.358,254.709,-110.940,171.132,42.143,158.043
C05247=1038.351,254.460,-110.911,171.130,42.142,158.042
C05248=1038.345,254.212,-110.881,171.126,42.141,158.042
C05249=1038.337,253.964,-110.853,171.124,42.140,158.041
C05250=1038.331,253.716,-110.823,171.120,42.139,158.041
C05251=1038.324,253.467,-110.793,171.118,42.137,158.041
C05252=1038.318,253.219,-110.764,171.114,42.136,158.040
C05253=1038.311,252.971,-110.735,171.112,42.135,158.040
C05254=1038.304,252.723,-110.705,171.109,42.133,158.039
C05255=1038.298,252.475,-110.676,171.106,42.132,158.039
C05256=1038.291,252.226,-110.647,171.103,42.131,158.038
C05257=1038.284,251.978,-110.618,171.100,42.130,158.038
C05258=1038.278,251.731,-110.588,171.097,42.129,158.037
C05259=1038.271,251.482,-110.559,171.094,42.127,158.037
C05260=1038.264,251.234,-110.530,171.091,42.126,158.036
C05261=1038.258,250.986,-110.501,171.089,42.125,158.036
C05262=1038.251,250.737,-110.472,171.085,42.123,158.035
C05263=1038.245,250.489,-110.443,171.082,42.122,158.035
C05264=1038.238,250.241,-110.413,171.079,42.121,158.034
C05265=1038.231,249.993,-110.384,171.076,42.119,158.034
C05266=1038.225,249.744,-110.355,171.074,42.118,158.034
C05267=1038.218,249.496,-110.326,171.070,42.117,158.033
C05268=1038.210,249.180,-110.288,171.067,42.116,158.033
C05269=1038.201,248.865,-110.252,171.063,42.114,158.032
C05270=1038.193,248.548,-110.215,171.059,42.112,158.031
C05271=1038.185,248.231,-110.177,171.056,42.111,158.031
C05272=1038.179,247.983,-110.148,171.053,42.109,158.030
C05273=1038.172,247.735,-110.119,171.050,42.108,158.030
C05274=1038.165,247.487,-110.091,171.047,42.107,158.029
C05275=1038.159,247.238,-110.061,171.044,42.105,158.029
C05276=1038.152,246.990,-110.032,171.041,42.105,158.029
C05277=1038.146,246.742,-110.003,171.038,42.103,158.028
C05278=1038.140,246.494,-109.974,171.036,42.101,158.028
C05279=1038.133,246.245,-109.945,171.032,42.101,158.027
C05280=1038.126,245.997,-109.916,171.030,42.099,158.027
C05281=1038.120,245.749,-109.887,171.027,42.098,158.026
C05282=1038.113,245.501,-109.858,171.025,42.097,158.026
C05283=1038.107,245.253,-109.829,171.021,42.095,158.025
C05284=1038.100,245.004,-109.800,171.019,42.094,158.025
C05285=1038.093,244.756,-109.771,171.016,42.093,158.024
C05286=1038.087,244.508,-109.742,171.013,42.092,158.024
C05287=1038.080,244.260,-109.714,171.010,42.090,158.023
C05288=1038.074,244.011,-109.685,171.008,42.089,158.023
C05289=1038.067,243.763,-109.656,171.004,42.088,158.023
C05290=1038.060,243.515,-109.628,171.002,42.087,158.022
C05291=1038.054,243.267,-109.599,170.999,42.085,158.022
C05292=1038.047,243.019,-109.570,170.996,42.085,158.021
C05293=1038.041,242.770,-109.541,170.993,42.083,158.021
C05294=1038.034,242.522,-109.513,170.991,42.082,158.020
C05295=1038.027,242.274,-109.484,170.987,42.081,158.020
C05296=1038.021,242.025,-109.455,170.985,42.080,158.020
C05297=1038.014,241.777,-109.427,170.982,42.078,158.019
C05298=1038.008,241.529,-109.398,170.979,42.077,158.019
C05299=1038.001,241.280,-109.369,170.976,42.076,158.018
C05300=1037.995,241.032,-109.341,170.974,42.075,158.018
C05301=1037.988,240.784,-109.313,170.971,42.073,158.017
C05302=1037.981,240.536,-109.284,170.968,42.073,158.017
C05303=1037.975,240.287,-109.256,170.965,42.072,158.017
C05304=1037.968,240.039,-109.227,170.963,42.070,158.016
C05305=1037.961,239.790,-109.199,170.959,42.069,158.016
C05306=1037.954,239.542,-109.170,170.957,42.068,158.015
C05307=1037.947,239.294,-109.142,170.954,42.067,158.015
C05308=1037.941,239.046,-109.113,170.952,42.066,158.014
C05309=1037.934,238.798,-109.085,170.948,42.064,158.014
C05310=1037.928,238.549,-109.057,170.946,42.063,158.014
C05311=1037.921,238.301,-109.028,170.943,42.062,158.013
C05312=1037.914,238.052,-109.000,170.940,42.061,158.013
C05313=1037.907,237.804,-108.972,170.938,42.060,158.012
C05314=1037.901,237.555,-108.943,170.935,42.059,158.012
C05315=1037.894,237.308,-108.915,170.933,42.058,158.011
C05316=1037.887,237.059,-108.887,170.929,42.057,158.011
C05317=1037.881,236.811,-108.859,170.927,42.055,158.011
C05318=1037.874,236.563,-108.830,170.924,42.054,158.010
C05319=1037.868,236.314,-108.803,170.922,42.053,158.010
C05320=1037.861,236.066,-108.774,170.918,42.052,158.009
C05321=1037.854,235.817,-108.746,170.916,42.051,158.009
C05322=1037.848,235.568,-108.718,170.913,42.049,158.008
C05323=1037.841,235.321,-108.689,170.911,42.049,158.008
C05324=1037.832,234.999,-108.653,170.907,42.047,158.008
C05325=1037.824,234.677,-108.617,170.904,42.046,158.007
C05326=1037.815,234.355,-108.580,170.900,42.044,158.007
C05327=1037.807,234.033,-108.544,170.896,42.043,158.006
C05328=1037.800,233.785,-108.516,170.894,42.042,158.006
C05329=1037.793,233.537,-108.488,170.891,42.040,158.005
C05330=1037.786,233.288,-108.459,170.888,42.039,158.005
C05331=1037.780,233.039,-108.431,170.885,42.038,158.004
C05332=1037.773,232.791,-108.403,170.883,42.037,158.004
C05333=1037.766,232.542,-108.376,170.881,42.036,158.004
C05334=1037.759,232.295,-108.347,170.878,42.034,158.003
C05335=1037.753,232.046,-108.319,170.875,42.034,158.003
C05336=1037.747,231.797,-108.291,170.872,42.033,158.002
C05337=1037.740,231.549,-108.263,170.870,42.031,158.002
C05338=1037.733,231.301,-108.235,170.867,42.030,158.001
C05339=1037.726,231.053,-108.207,170.865,42.029,158.001
C05340=1037.720,230.804,-108.179,170.862,42.028,158.001
C05341=1037.714,230.556,-108.152,170.859,42.027,158.000
C05342=1037.707,230.308,-108.124,170.857,42.026,158.000
C05343=1037.701,230.059,-108.096,170.854,42.024,157.999
C05344=1037.694,229.811,-108.068,170.852,42.023,157.999
C05345=1037.688,229.562,-108.041,170.849,42.022,157.999
C05346=1037.681,229.315,-108.012,170.847,42.021,157.998
C05347=1037.674,229.066,-107.984,170.843,42.020,157.998
C05348=1037.667,228.818,-107.957,170.841,42.019,157.997
C05349=1037.661,228.569,-107.929,170.838,42.018,157.997
C05350=1037.654,228.321,-107.901,170.836,42.017,157.997
C05351=1037.647,228.072,-107.873,170.833,42.016,157.996
C05352=1037.641,227.824,-107.846,170.831,42.015,157.996
C05353=1037.634,227.575,-107.818,170.828,42.014,157.995
C05354=1037.627,227.327,-107.790,170.825,42.012,157.995
C05355=1037.620,227.079,-107.763,170.823,42.011,157.995
C05356=1037.613,226.830,-107.735,170.820,42.010,157.994
C05357=1037.606,226.582,-107.708,170.818,42.009,157.994
C05358=1037.600,226.333,-107.681,170.815,42.008,157.994
C05359=1037.593,226.085,-107.653,170.812,42.007,157.993
C05360=1037.587,225.836,-107.625,170.809,42.006,157.993
C05361=1037.580,225.588,-107.597,170.807,42.005,157.992
C05362=1037.573,225.340,-107.571,170.805,42.004,157.992
C05363=1037.567,225.092,-107.543,170.802,42.003,157.991
C05364=1037.560,224.843,-107.515,170.800,42.002,157.991
C05365=1037.553,224.595,-107.488,170.797,42.001,157.991
C05366=1037.547,224.346,-107.461,170.795,42.000,157.990
C05367=1037.540,224.097,-107.433,170.791,41.999,157.990
C05368=1037.533,223.849,-107.406,170.789,41.997,157.989
C05369=1037.526,223.601,-107.378,170.786,41.996,157.989
C05370=1037.519,223.352,-107.350,170.784,41.995,157.989
C05371=1037.513,223.105,-107.323,170.782,41.994,157.988
C05372=1037.507,222.856,-107.296,170.779,41.993,157.988
C05373=1037.500,222.607,-107.268,170.777,41.992,157.988
C05374=1037.493,222.359,-107.241,170.774,41.991,157.987
C05375=1037.486,222.111,-107.213,170.772,41.990,157.987
C05376=1037.480,221.861,-107.186,170.769,41.988,157.986
C05377=1037.474,221.614,-107.159,170.766,41.988,157.986
C05378=1037.467,221.365,-107.131,170.763,41.987,157.986
C05379=1037.460,221.117,-107.103,170.761,41.986,157.985
C05380=1037.452,220.787,-107.068,170.758,41.984,157.985
C05381=1037.443,220.458,-107.032,170.755,41.983,157.984
C05382=1037.434,220.128,-106.995,170.751,41.981,157.984
C05383=1037.425,219.799,-106.959,170.748,41.980,157.983
C05384=1037.418,219.550,-106.931,170.745,41.979,157.983
C05385=1037.411,219.302,-106.905,170.743,41.978,157.982
C05386=1037.405,219.054,-106.878,170.740,41.977,157.982
C05387=1037.398,218.805,-106.851,170.738,41.975,157.982
C05388=1037.391,218.557,-106.823,170.735,41.974,157.981
C05389=1037.384,218.308,-106.797,170.733,41.973,157.981
C05390=1037.378,218.060,-106.769,170.731,41.973,157.981
C05391=1037.370,217.811,-106.742,170.728,41.972,157.980
C05392=1037.364,217.563,-106.716,170.726,41.971,157.980
C05393=1037.358,217.315,-106.688,170.724,41.970,157.980
C05394=1037.351,217.066,-106.661,170.721,41.968,157.979
C05395=1037.344,216.817,-106.634,170.719,41.967,157.979
